KUKA KRL program: MyProgram_202().src

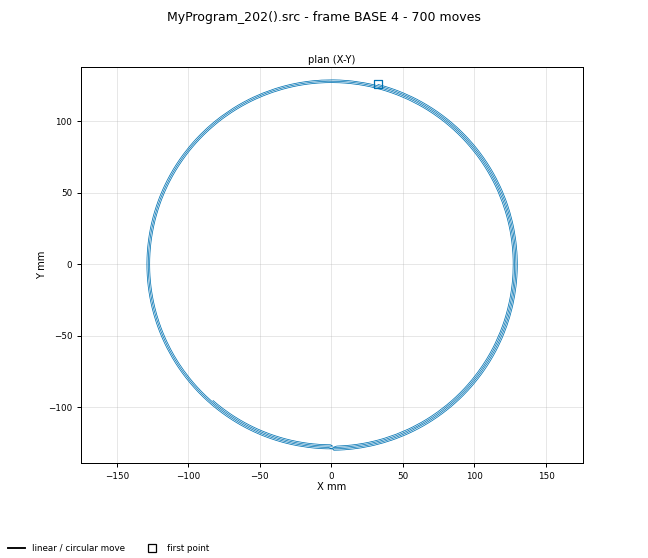
[picture p0: tool path of MyProgram_202().src in frame BASE 4, 700 of 700 moves have a stored position in this frame; points joined in program order, loops and branches not executed]
&ACCESS RVP
&REL 1
&PARAM TEMPLATE = C:\KRC\Roboter\Template\vorgabe
&PARAM EDITMASK = *
DEF MyProgram_202()
; ---- Setting reference (Base) ----
$BASE = BASE_DATA[4]

; --------------------------
; ---- Setting tool (TCP) ----
$TOOL = TOOL_DATA[3]
; --------------------------

$VEL.CP = VEL_APROX_PRINT
Startdeposition()
$VEL.CP = VEL_PRINT
LIN {X 32.4912,Y 125.808,Z 145,A 71.2576,B 24.9481,C -1.6638,E1 25.0411,E2 735.1147} C_DIS
LIN {X 35.4969,Y 124.993,Z 145,A 69.8884,B 24.9481,C -1.663,E1 25.0447,E2 736.4834} C_DIS
LIN {X 38.2252,Y 124.1849,Z 145,A 68.5665,B 24.9484,C -1.6587,E1 25.0483,E2 737.8133} C_DIS
LIN {X 41.3157,Y 123.1913,Z 145,A 67.1752,B 24.9484,C -1.6595,E1 25.052,E2 739.1999} C_DIS
LIN {X 44.3236,Y 122.1413,Z 145,A 65.7721,B 24.9484,C -1.6583,E1 25.0557,E2 740.6031} C_DIS
LIN {X 47.3297,Y 121.0081,Z 145,A 64.3243,B 24.9487,C -1.6553,E1 25.0595,E2 742.0548} C_DIS
LIN {X 50.4558,Y 119.7388,Z 145,A 62.8585,B 24.9487,C -1.6548,E1 25.0632,E2 743.5183} C_DIS
LIN {X 53.4411,Y 118.4365,Z 145,A 61.4515,B 24.9487,C -1.6547,E1 25.0668,E2 744.9223} C_DIS
LIN {X 56.2396,Y 117.133,Z 145,A 60.0583,B 24.9489,C -1.6514,E1 25.0703,E2 746.3197} C_DIS
LIN {X 59.4678,Y 115.5287,Z 145,A 58.4153,B 24.9492,C -1.6465,E1 25.0745,E2 747.9697} C_DIS
LIN {X 63.2279,Y 113.5157,Z 145,A 56.501,B 24.9495,C -1.6421,E1 25.0792,E2 749.8887} C_DIS
LIN {X 66.9845,Y 111.3401,Z 145,A 54.5775,B 24.9497,C -1.6388,E1 25.0838,E2 751.8143} C_DIS
LIN {X 70.8468,Y 108.923,Z 145,A 52.626,B 24.9497,C -1.6385,E1 25.0884,E2 753.76} C_DIS
LIN {X 74.4541,Y 106.4901,Z 145,A 50.7053,B 24.9499,C -1.6352,E1 25.0928,E2 755.6822} C_DIS
LIN {X 77.9363,Y 103.9691,Z 145,A 48.7841,B 24.9502,C -1.6304,E1 25.0971,E2 757.6077} C_DIS
LIN {X 81.3309,Y 101.3353,Z 145,A 46.8925,B 24.9504,C -1.627,E1 25.1013,E2 759.5003} C_DIS
LIN {X 84.4776,Y 98.7278,Z 145,A 45.1201,B 24.9505,C -1.625,E1 25.1051,E2 761.2706} C_DIS
LIN {X 87.6247,Y 95.9456,Z 145,A 43.3009,B 24.9506,C -1.6229,E1 25.1088,E2 763.0875} C_DIS
LIN {X 90.595,Y 93.1456,Z 145,A 41.5081,B 24.9509,C -1.6195,E1 25.1124,E2 764.881} C_DIS
LIN {X 93.6458,Y 90.0783,Z 145,A 39.6489,B 24.9509,C -1.6178,E1 25.1161,E2 766.7363} C_DIS
LIN {X 96.4286,Y 87.0923,Z 145,A 37.8481,B 24.9512,C -1.6136,E1 25.1195,E2 768.539} C_DIS
LIN {X 99.1768,Y 83.9494,Z 145,A 36.042,B 24.9514,C -1.6111,E1 25.1228,E2 770.3429} C_DIS
LIN {X 101.4035,Y 81.2464,Z 145,A 34.4908,B 24.9516,C -1.607,E1 25.1255,E2 771.8966} C_DIS
LIN {X 103.8668,Y 78.0719,Z 145,A 32.6881,B 24.952,C -1.6009,E1 25.1286,E2 773.705} C_DIS
LIN {X 106.4211,Y 74.5532,Z 145,A 30.7475,B 24.9523,C -1.5948,E1 25.1317,E2 775.6507} C_DIS
LIN {X 108.7748,Y 71.075,Z 145,A 28.8761,B 24.9527,C -1.5889,E1 25.1346,E2 777.5267} C_DIS
LIN {X 111.0977,Y 67.3855,Z 145,A 27.0107,B 24.9528,C -1.5867,E1 25.1374,E2 779.3877} C_DIS
LIN {X 113.2935,Y 63.6243,Z 145,A 25.1416,B 24.953,C -1.5841,E1 25.14,E2 781.2532} C_DIS
LIN {X 115.2071,Y 60.0868,Z 145,A 23.4203,B 24.9531,C -1.5819,E1 25.1422,E2 782.9706} C_DIS
LIN {X 116.7275,Y 57.0777,Z 145,A 21.9744,B 24.9532,C -1.5798,E1 25.144,E2 784.4138} C_DIS
LIN {X 118.0523,Y 54.2836,Z 145,A 20.5723,B 24.9536,C -1.5738,E1 25.1457,E2 785.8224} C_DIS
LIN {X 119.393,Y 51.2678,Z 145,A 19.1594,B 24.9537,C -1.5718,E1 25.1472,E2 787.2323} C_DIS
LIN {X 120.7266,Y 48.0458,Z 145,A 17.6476,B 24.9539,C -1.5686,E1 25.1488,E2 788.7434} C_DIS
LIN {X 121.789,Y 45.2829,Z 145,A 16.3455,B 24.9541,C -1.5649,E1 25.1501,E2 790.0471} C_DIS
LIN {X 122.9304,Y 42.0878,Z 145,A 14.8729,B 24.9543,C -1.5615,E1 25.1515,E2 791.5193} C_DIS
LIN {X 124.0143,Y 38.7826,Z 145,A 13.332,B 24.9546,C -1.5564,E1 25.1528,E2 793.0634} C_DIS
LIN {X 124.7733,Y 36.2591,Z 145,A 12.1683,B 24.9548,C -1.5528,E1 25.1537,E2 794.2291} C_DIS
LIN {X 125.6228,Y 33.1968,Z 145,A 10.7859,B 24.955,C -1.5494,E1 25.1547,E2 795.6116} C_DIS
LIN {X 126.3733,Y 30.2137,Z 145,A 9.4857,B 24.955,C -1.5481,E1 25.1556,E2 796.9072} C_DIS
LIN {X 127.0123,Y 27.403,Z 145,A 8.1592,B 24.9555,C -1.5411,E1 25.1564,E2 798.2425} C_DIS
LIN {X 127.6864,Y 24.0695,Z 145,A 6.6754,B 24.9557,C -1.5372,E1 25.1572,E2 799.727} C_DIS
LIN {X 128.2522,Y 20.8498,Z 145,A 5.2557,B 24.9559,C -1.5337,E1 25.1579,E2 801.1466} C_DIS
LIN {X 128.7042,Y 17.8487,Z 145,A 3.9702,B 24.956,C -1.5322,E1 25.1584,E2 802.428} C_DIS
LIN {X 129.0189,Y 15.4011,Z 145,A 2.831,B 24.9564,C -1.5259,E1 25.1588,E2 803.5752} C_DIS
LIN {X 129.3909,Y 11.89,Z 145,A 1.3171,B 24.9565,C -1.5231,E1 25.1592,E2 805.0868} C_DIS
LIN {X 129.6283,Y 8.9369,Z 145,A 0.0617,B 24.9566,C -1.5216,E1 25.1595,E2 806.3383} C_DIS
LIN {X 129.7846,Y 6.2559,Z 145,A -1.1949,B 24.9571,C -1.5138,E1 25.1596,E2 807.6058} C_DIS
LIN {X 129.9157,Y 2.2459,Z 145,A -2.9323,B 24.9573,C -1.5097,E1 25.1598,E2 809.3425} C_DIS
LIN {X 129.9256,Y -1.648,Z 145,A -4.7087,B 24.9578,C -1.5008,E1 25.1598,E2 811.1293} C_DIS
LIN {X 129.8316,Y -5.1857,Z 145,A -6.2154,B 24.9579,C -1.4986,E1 25.1596,E2 812.6323} C_DIS
LIN {X 129.6439,Y -8.7237,Z 145,A -7.7185,B 24.958,C -1.4966,E1 25.1594,E2 814.1312} C_DIS
LIN {X 129.3753,Y -12.0517,Z 145,A -9.2549,B 24.9585,C -1.4883,E1 25.159,E2 815.678} C_DIS
LIN {X 129.012,Y -15.4589,Z 145,A -10.7277,B 24.9587,C -1.4853,E1 25.1585,E2 817.1491} C_DIS
LIN {X 128.5211,Y -19.1304,Z 145,A -12.3114,B 24.9588,C -1.4826,E1 25.1579,E2 818.73} C_DIS
LIN {X 128.0736,Y -21.9207,Z 145,A -13.5064,B 24.9588,C -1.4813,E1 25.1574,E2 819.9211} C_DIS
LIN {X 127.6134,Y -24.4517,Z 145,A -14.6895,B 24.9592,C -1.4749,E1 25.1568,E2 821.1122} C_DIS
LIN {X 126.9339,Y -27.7659,Z 145,A -16.1647,B 24.9595,C -1.4709,E1 25.1559,E2 822.5881} C_DIS
LIN {X 126.2492,Y -30.7286,Z 145,A -17.4909,B 24.9597,C -1.4673,E1 25.1551,E2 823.9151} C_DIS
LIN {X 125.4352,Y -33.9003,Z 145,A -18.9313,B 24.9599,C -1.4628,E1 25.154,E2 825.3578} C_DIS
LIN {X 124.6228,Y -36.7728,Z 145,A -20.2611,B 24.9602,C -1.4579,E1 25.153,E2 826.6918} C_DIS
LIN {X 123.6135,Y -40.0371,Z 145,A -21.7437,B 24.9604,C -1.4543,E1 25.1518,E2 828.1744} C_DIS
LIN {X 122.6529,Y -42.888,Z 145,A -23.0454,B 24.9605,C -1.4514,E1 25.1506,E2 829.4756} C_DIS
LIN {X 121.5617,Y -45.8895,Z 145,A -24.4397,B 24.9607,C -1.4477,E1 25.1492,E2 830.8707} C_DIS
LIN {X 120.4111,Y -48.8285,Z 145,A -25.8611,B 24.9611,C -1.4417,E1 25.1478,E2 832.2984} C_DIS
LIN {X 119.0356,Y -52.0946,Z 145,A -27.3824,B 24.9612,C -1.439,E1 25.1461,E2 833.8176} C_DIS
LIN {X 117.594,Y -55.2747,Z 145,A -28.9303,B 24.9615,C -1.4338,E1 25.1443,E2 835.3695} C_DIS
LIN {X 116.4176,Y -57.7059,Z 145,A -30.1387,B 24.9617,C -1.4293,E1 25.1428,E2 836.5822} C_DIS
LIN {X 115.017,Y -60.4488,Z 145,A -31.4457,B 24.9618,C -1.4279,E1 25.1411,E2 837.8855} C_DIS
LIN {X 113.0688,Y -64.0241,Z 145,A -33.3523,B 24.9624,C -1.4165,E1 25.1385,E2 839.809} C_DIS
LIN {X 110.9386,Y -67.6478,Z 145,A -35.2233,B 24.9628,C -1.4101,E1 25.1358,E2 841.6854} C_DIS
LIN {X 108.7567,Y -71.1028,Z 145,A -36.8864,B 24.9626,C -1.4123,E1 25.1333,E2 843.3351} C_DIS
LIN {X 106.8976,Y -73.8683,Z 145,A -38.3473,B 24.9628,C -1.4086,E1 25.131,E2 844.7976} C_DIS
LIN {X 104.8526,Y -76.7427,Z 145,A -39.995,B 24.9633,C -1.3993,E1 25.1283,E2 846.4591} C_DIS
LIN {X 102.2417,Y -80.1879,Z 145,A -41.8596,B 24.9635,C -1.3962,E1 25.1251,E2 848.3222} C_DIS
LIN {X 99.8885,Y -83.1014,Z 145,A -43.4331,B 24.9635,C -1.3959,E1 25.1224,E2 849.889} C_DIS
LIN {X 97.7073,Y -85.6553,Z 145,A -44.9059,B 24.9637,C -1.3925,E1 25.1197,E2 851.3634} C_DIS
LIN {X 95.2327,Y -88.3982,Z 145,A -46.6386,B 24.9642,C -1.3827,E1 25.1164,E2 853.1114} C_DIS
LIN {X 92.0534,Y -91.7042,Z 145,A -48.5566,B 24.9642,C -1.3832,E1 25.1126,E2 855.0202} C_DIS
LIN {X 89.4704,Y -94.2268,Z 145,A -50.1556,B 24.9644,C -1.3789,E1 25.1094,E2 856.6226} C_DIS
LIN {X 86.4321,Y -97.021,Z 145,A -52.0108,B 24.9647,C -1.3727,E1 25.1056,E2 858.485} C_DIS
LIN {X 83.2465,Y -99.7678,Z 145,A -53.7858,B 24.9647,C -1.3727,E1 25.1018,E2 860.2532} C_DIS
LIN {X 80.5905,Y -101.9255,Z 145,A -55.2797,B 24.9648,C -1.37,E1 25.0986,E2 861.7477} C_DIS
LIN {X 77.5468,Y -104.2591,Z 145,A -57.0149,B 24.9651,C -1.364,E1 25.0947,E2 863.4907} C_DIS
LIN {X 74.0334,Y -106.7828,Z 145,A -58.9095,B 24.9653,C -1.3607,E1 25.0903,E2 865.3865} C_DIS
LIN {X 70.5061,Y -109.1441,Z 145,A -60.7379,B 24.9653,C -1.3592,E1 25.0861,E2 867.2124} C_DIS
LIN {X 67.5911,Y -110.9734,Z 145,A -62.3516,B 24.9658,C -1.3512,E1 25.0822,E2 868.8399} C_DIS
LIN {X 63.857,Y -113.1627,Z 145,A -64.2476,B 24.9659,C -1.3484,E1 25.0776,E2 870.7369} C_DIS
LIN {X 59.89,Y -115.3104,Z 145,A -66.1258,B 24.9659,C -1.3507,E1 25.073,E2 872.6042} C_DIS
LIN {X 57.2655,Y -116.6348,Z 145,A -67.4291,B 24.9659,C -1.3482,E1 25.0698,E2 873.91} C_DIS
LIN {X 54.009,Y -118.1792,Z 145,A -68.987,B 24.966,C -1.3473,E1 25.0658,E2 875.4662} C_DIS
LIN {X 51.1346,Y -119.4506,Z 145,A -70.3453,B 24.966,C -1.3466,E1 25.0624,E2 876.8227} C_DIS
LIN {X 48.119,Y -120.6971,Z 145,A -71.7959,B 24.9662,C -1.3439,E1 25.0586,E2 878.2764} C_DIS
LIN {X 45.203,Y -121.8189,Z 145,A -73.1449,B 24.9662,C -1.3435,E1 25.0551,E2 879.6235} C_DIS
LIN {X 42.4199,Y -122.8152,Z 145,A -74.4837,B 24.9664,C -1.3399,E1 25.0515,E2 880.968} C_DIS
LIN {X 39.0302,Y -123.9352,Z 145,A -76.0399,B 24.9664,C -1.3389,E1 25.0474,E2 882.5237} C_DIS
LIN {X 36.2163,Y -124.7858,Z 145,A -77.3172,B 24.9664,C -1.3384,E1 25.044,E2 883.8} C_DIS
LIN {X 33.1812,Y -125.6269,Z 145,A -78.7387,B 24.9666,C -1.3352,E1 25.0401,E2 885.2268} C_DIS
LIN {X 30.2349,Y -126.3682,Z 145,A -80.0521,B 24.9666,C -1.3352,E1 25.0366,E2 886.5383} C_DIS
LIN {X 27.2585,Y -127.0435,Z 145,A -81.4363,B 24.9668,C -1.3319,E1 25.0328,E2 887.9283} C_DIS
LIN {X 23.6437,Y -127.7678,Z 145,A -83.0096,B 24.9668,C -1.3332,E1 25.0285,E2 889.4968} C_DIS
LIN {X 20.8498,Y -128.2522,Z 145,A -84.2663,B 24.9668,C -1.3319,E1 25.025,E2 890.7552} C_DIS
LIN {X 17.8487,Y -128.7042,Z 145,A -85.6004,B 24.9668,C -1.3312,E1 25.0213,E2 892.0898} C_DIS
LIN {X 14.8613,Y -129.0833,Z 145,A -86.924,B 24.9668,C -1.3306,E1 25.0177,E2 893.4139} C_DIS
LIN {X 11.89,Y -129.3909,Z 145,A -88.192,B 24.9668,C -1.3324,E1 25.0142,E2 894.6769} C_DIS
LIN {X 9.2153,Y -129.608,Z 145,A -89.4167,B 24.9668,C -1.3297,E1 25.0107,E2 895.9073} C_DIS
LIN {X 5.3463,Y -129.8253,Z 145,A -91.179,B 24.9671,C -1.3263,E1 25.0058,E2 897.6771} C_DIS
LIN {X 1.648,Y -129.9256,Z 145,A -92.7481,B 24.9669,C -1.3289,E1 25.0014,E2 899.2396} C_DIS
LIN {X 1.648,Y -129.9256,Z 145,A -92.7481,B 24.9669,C -1.3289,E1 25.0014,E2 899.2396} C_DIS
Enddeposition()
LIN {X 0.9172,Y -128.9653,Z 145,A -92.8374,B 24.5098,C -1.2621,E1 24.5412,E2 899.4275} C_DIS
Startdeposition()
$VEL.CP = VEL_PRINT
LIN {X 5.042,Y -128.8762,Z 145,A -90.5283,B 24.5086,C -1.2863,E1 24.5478,E2 897.0606} C_DIS
LIN {X 8.2974,Y -128.7081,Z 145,A -88.9865,B 24.5084,C -1.2916,E1 24.5521,E2 895.5066} C_DIS
LIN {X 12.5181,Y -128.3659,Z 145,A -87.1558,B 24.5084,C -1.29,E1 24.5572,E2 893.6807} C_DIS
LIN {X 18.1324,Y -127.6937,Z 145,A -84.5266,B 24.5081,C -1.2976,E1 24.5645,E2 891.0355} C_DIS
LIN {X 22.5529,Y -126.9876,Z 145,A -82.639,B 24.5083,C -1.294,E1 24.5697,E2 889.1586} C_DIS
LIN {X 26.1324,Y -126.3001,Z 145,A -80.9242,B 24.5079,C -1.3002,E1 24.5744,E2 887.4308} C_DIS
LIN {X 30.1447,Y -125.4023,Z 145,A -79.2248,B 24.5082,C -1.2955,E1 24.579,E2 885.7451} C_DIS
LIN {X 33.3745,Y -124.5816,Z 145,A -77.7418,B 24.5081,C -1.2972,E1 24.583,E2 884.2605} C_DIS
LIN {X 37.1134,Y -123.521,Z 145,A -75.7574,B 24.5073,C -1.3124,E1 24.5884,E2 882.2431} C_DIS
LIN {X 42.3908,Y -121.809,Z 145,A -73.5836,B 24.5079,C -1.3006,E1 24.5941,E2 880.1019} C_DIS
LIN {X 45.7996,Y -120.5701,Z 145,A -71.8309,B 24.5075,C -1.31,E1 24.5987,E2 878.3304} C_DIS
LIN {X 49.5713,Y -119.0676,Z 145,A -69.8378,B 24.5068,C -1.3224,E1 24.6039,E2 876.3122} C_DIS
LIN {X 52.6398,Y -117.743,Z 145,A -68.6461,B 24.5075,C -1.3096,E1 24.6069,E2 875.1542} C_DIS
LIN {X 56.4236,Y -115.9795,Z 145,A -66.7297,B 24.5072,C -1.3157,E1 24.6118,E2 873.2281} C_DIS
LIN {X 65.6898,Y -110.9946,Z 145,A -62.1749,B 24.5071,C -1.3177,E1 24.6229,E2 868.6821} C_DIS
LIN {X 69.8564,Y -108.4208,Z 145,A -60.0132,B 24.5069,C -1.3212,E1 24.628,E2 866.5192} C_DIS
LIN {X 72.8158,Y -106.4554,Z 145,A -58.3755,B 24.5066,C -1.3275,E1 24.6318,E2 864.8719} C_DIS
LIN {X 76.1855,Y -104.0705,Z 145,A -56.501,B 24.5063,C -1.3334,E1 24.6361,E2 862.9898} C_DIS
LIN {X 79.4416,Y -101.6069,Z 145,A -54.6674,B 24.506,C -1.3384,E1 24.6401,E2 861.1511} C_DIS
LIN {X 82.3725,Y -99.2453,Z 145,A -53.098,B 24.506,C -1.3368,E1 24.6435,E2 859.5916} C_DIS
LIN {X 85.2992,Y -96.7416,Z 145,A -51.4153,B 24.506,C -1.3393,E1 24.647,E2 857.9097} C_DIS
LIN {X 88.2732,Y -94.0361,Z 145,A -49.5828,B 24.5056,C -1.3461,E1 24.6508,E2 856.0687} C_DIS
LIN {X 91.1569,Y -91.2436,Z 145,A -47.9186,B 24.5057,C -1.3442,E1 24.6541,E2 854.416} C_DIS
LIN {X 93.7338,Y -88.5936,Z 145,A -46.1682,B 24.5052,C -1.354,E1 24.6575,E2 852.6497} C_DIS
LIN {X 96.647,Y -85.4061,Z 145,A -44.3102,B 24.5052,C -1.3558,E1 24.661,E2 850.7959} C_DIS
LIN {X 99.348,Y -82.2485,Z 145,A -42.3389,B 24.5045,C -1.3674,E1 24.6646,E2 848.8061} C_DIS
LIN {X 102.2616,Y -78.5971,Z 145,A -40.3258,B 24.5044,C -1.3697,E1 24.668,E2 846.7971} C_DIS
LIN {X 104.9015,Y -75.0369,Z 145,A -38.2409,B 24.5038,C -1.3814,E1 24.6715,E2 844.6946} C_DIS
LIN {X 109.1864,Y -68.6522,Z 145,A -34.9427,B 24.5036,C -1.3849,E1 24.6765,E2 841.4047} C_DIS
LIN {X 111.0541,Y -65.5892,Z 145,A -33.3576,B 24.5034,C -1.3891,E1 24.6788,E2 839.8179} C_DIS
LIN {X 113.3781,Y -61.4847,Z 145,A -31.3272,B 24.5032,C -1.3919,E1 24.6815,E2 837.7915} C_DIS
LIN {X 115.0369,Y -58.3174,Z 145,A -29.8444,B 24.5032,C -1.3911,E1 24.6834,E2 836.3185} C_DIS
LIN {X 116.7701,Y -54.7687,Z 145,A -27.7093,B 24.5019,C -1.4167,E1 24.686,E2 834.1339} C_DIS
LIN {X 118.2649,Y -51.4575,Z 145,A -26.7258,B 24.5034,C -1.3883,E1 24.687,E2 833.2241} C_DIS
LIN {X 119.0606,Y -49.588,Z 145,A -25.6136,B 24.5027,C -1.4022,E1 24.6883,E2 832.0848} C_DIS
LIN {X 120.3938,Y -46.2598,Z 145,A -23.9046,B 24.5021,C -1.4133,E1 24.69,E2 830.3587} C_DIS
LIN {X 122.2439,Y -41.1214,Z 145,A -21.7994,B 24.5026,C -1.404,E1 24.6919,E2 828.2879} C_DIS
LIN {X 123.0704,Y -38.5821,Z 145,A -20.2512,B 24.5013,C -1.4269,E1 24.6933,E2 826.6937} C_DIS
LIN {X 124.2424,Y -34.6157,Z 145,A -18.6205,B 24.5016,C -1.4219,E1 24.6945,E2 825.0846} C_DIS
LIN {X 125.2378,Y -30.8269,Z 145,A -16.794,B 24.501,C -1.4321,E1 24.6958,E2 823.2445} C_DIS
LIN {X 126.0851,Y -27.1474,Z 145,A -15.2551,B 24.5011,C -1.4302,E1 24.6967,E2 821.7191} C_DIS
LIN {X 126.7255,Y -23.982,Z 145,A -13.7893,B 24.5008,C -1.4366,E1 24.6975,E2 820.2469} C_DIS
LIN {X 127.4291,Y -19.9072,Z 145,A -10.7727,B 24.4969,C -1.5058,E1 24.6989,E2 817.0823} C_DIS
LIN {X 128.4003,Y -12.1599,Z 145,A -8.7524,B 24.5006,C -1.4396,E1 24.6994,E2 815.233} C_DIS
LIN {X 128.6857,Y -8.6592,Z 145,A -6.7679,B 24.4991,C -1.4672,E1 24.6998,E2 813.1944} C_DIS
LIN {X 128.9118,Y -4.058,Z 145,A -4.8212,B 24.4991,C -1.4686,E1 24.7,E2 811.2561} C_DIS
LIN {X 128.9762,Y 0.3437,Z 145,A -2.8995,B 24.4988,C -1.4732,E1 24.7,E2 809.3351} C_DIS
LIN {X 128.758,Y 7.4881,Z 145,A 0.0508,B 24.4988,C -1.4717,E1 24.6998,E2 806.4064} C_DIS
LIN {X 128.2242,Y 13.8938,Z 145,A 3.0101,B 24.498,C -1.4864,E1 24.699,E2 803.4297} C_DIS
LIN {X 127.7263,Y 17.9044,Z 145,A 4.5867,B 24.4983,C -1.4806,E1 24.6985,E2 801.8765} C_DIS
LIN {X 127.3111,Y 20.6556,Z 145,A 6.0944,B 24.4973,C -1.4989,E1 24.6978,E2 800.3339} C_DIS
LIN {X 126.6844,Y 24.1973,Z 145,A 7.5774,B 24.4973,C -1.498,E1 24.697,E2 798.862} C_DIS
LIN {X 125.9668,Y 27.6953,Z 145,A 9.2816,B 24.4967,C -1.5092,E1 24.696,E2 797.141} C_DIS
LIN {X 125.0296,Y 31.6546,Z 145,A 10.9355,B 24.4968,C -1.5068,E1 24.6949,E2 795.5027} C_DIS
LIN {X 124.1886,Y 34.8083,Z 145,A 12.3832,B 24.4966,C -1.5112,E1 24.6939,E2 794.0529} C_DIS
LIN {X 123.1959,Y 38.1755,Z 145,A 14.0747,B 24.4959,C -1.523,E1 24.6925,E2 792.3431} C_DIS
LIN {X 121.8051,Y 42.402,Z 145,A 15.9011,B 24.496,C -1.5211,E1 24.6909,E2 790.5318} C_DIS
LIN {X 120.7475,Y 45.3258,Z 145,A 17.277,B 24.4958,C -1.5249,E1 24.6895,E2 789.1544} C_DIS
LIN {X 119.3674,Y 48.8493,Z 145,A 19.2308,B 24.4946,C -1.5443,E1 24.6875,E2 787.1653} C_DIS
LIN {X 117.5648,Y 53.0382,Z 145,A 20.9232,B 24.4953,C -1.5327,E1 24.6856,E2 785.5102} C_DIS
LIN {X 116.3389,Y 55.6743,Z 145,A 22.2306,B 24.4951,C -1.5372,E1 24.684,E2 784.199} C_DIS
LIN {X 114.7641,Y 58.8533,Z 145,A 23.8574,B 24.4946,C -1.5443,E1 24.682,E2 782.564} C_DIS
LIN {X 112.6959,Y 62.7261,Z 145,A 25.9472,B 24.4939,C -1.557,E1 24.6791,E2 780.4549} C_DIS
LIN {X 110.1549,Y 67.0888,Z 145,A 28.1143,B 24.4938,C -1.5592,E1 24.6761,E2 778.294} C_DIS
LIN {X 108.2811,Y 70.072,Z 145,A 29.6406,B 24.4936,C -1.5613,E1 24.6738,E2 776.7705} C_DIS
LIN {X 105.8567,Y 73.6831,Z 145,A 31.5435,B 24.4934,C -1.5648,E1 24.6708,E2 774.8688} C_DIS
LIN {X 103.2464,Y 77.2991,Z 145,A 33.4979,B 24.4932,C -1.5684,E1 24.6675,E2 772.9154} C_DIS
LIN {X 100.8045,Y 80.4571,Z 145,A 35.2068,B 24.4932,C -1.5694,E1 24.6646,E2 771.2121} C_DIS
LIN {X 98.543,Y 83.2124,Z 145,A 36.8806,B 24.4926,C -1.5779,E1 24.6616,E2 769.5259} C_DIS
LIN {X 95.7514,Y 86.4097,Z 145,A 39.3329,B 24.4906,C -1.6117,E1 24.6569,E2 767.0034} C_DIS
LIN {X 92.2184,Y 90.1699,Z 145,A 40.9534,B 24.4924,C -1.5819,E1 24.6539,E2 765.4616} C_DIS
LIN {X 89.338,Y 93.0251,Z 145,A 42.8345,B 24.4919,C -1.5899,E1 24.6501,E2 763.5695} C_DIS
LIN {X 86.0756,Y 96.0512,Z 145,A 44.7867,B 24.4917,C -1.5927,E1 24.6461,E2 761.6186} C_DIS
LIN {X 82.823,Y 98.8697,Z 145,A 46.6014,B 24.4918,C -1.5915,E1 24.6422,E2 759.814} C_DIS
LIN {X 79.9093,Y 101.2395,Z 145,A 48.3383,B 24.4914,C -1.5981,E1 24.6384,E2 758.0677} C_DIS
LIN {X 76.5354,Y 103.8134,Z 145,A 50.2418,B 24.4911,C -1.6025,E1 24.6342,E2 756.1607} C_DIS
LIN {X 73.1048,Y 106.257,Z 145,A 52.1163,B 24.4909,C -1.6059,E1 24.6299,E2 754.2848} C_DIS
LIN {X 69.2727,Y 108.7945,Z 145,A 54.192,B 24.4906,C -1.6109,E1 24.625,E2 752.2039} C_DIS
LIN {X 65.331,Y 111.2057,Z 145,A 56.2125,B 24.4906,C -1.6124,E1 24.6202,E2 750.1862} C_DIS
LIN {X 61.4184,Y 113.4143,Z 145,A 58.1643,B 24.4905,C -1.613,E1 24.6154,E2 748.2388} C_DIS
LIN {X 58.3822,Y 115.0039,Z 145,A 59.5685,B 24.4907,C -1.609,E1 24.6119,E2 746.8481} C_DIS
LIN {X 55.3148,Y 116.5107,Z 145,A 61.0639,B 24.4907,C -1.6098,E1 24.6082,E2 745.3548} C_DIS
LIN {X 52.5043,Y 117.8036,Z 145,A 62.4741,B 24.4905,C -1.6132,E1 24.6046,E2 743.94} C_DIS
LIN {X 48.9828,Y 119.3133,Z 145,A 64.142,B 24.4905,C -1.6133,E1 24.6003,E2 742.2758} C_DIS
LIN {X 45.0791,Y 120.8399,Z 145,A 66.0297,B 24.4903,C -1.6165,E1 24.5954,E2 740.3847} C_DIS
LIN {X 41.5737,Y 122.0923,Z 145,A 67.8767,B 24.4896,C -1.6276,E1 24.5904,E2 738.5146} C_DIS
LIN {X 37.3576,Y 123.4462,Z 145,A 69.6419,B 24.4901,C -1.6191,E1 24.5858,E2 736.7733} C_DIS
LIN {X 33.4874,Y 124.5515,Z 145,A 71.4784,B 24.4899,C -1.6227,E1 24.5808,E2 734.9311} C_DIS
LIN {X 30.2084,Y 125.3869,Z 145,A 72.9173,B 24.49,C -1.6205,E1 24.577,E2 733.4998} C_DIS
LIN {X 26.7242,Y 126.1765,Z 145,A 74.6365,B 24.4896,C -1.6278,E1 24.5722,E2 731.7653} C_DIS
LIN {X 22.7495,Y 126.9524,Z 145,A 76.3137,B 24.4899,C -1.6225,E1 24.5677,E2 730.1026} C_DIS
LIN {X 14.6498,Y 128.1407,Z 145,A 79.8929,B 24.49,C -1.6205,E1 24.5578,E2 726.5314} C_DIS
LIN {X 11.5908,Y 128.4549,Z 145,A 82.1032,B 24.4874,C -1.6624,E1 24.5514,E2 724.2215} C_DIS
LIN {X 5.9542,Y 128.8383,Z 145,A 83.6204,B 24.4905,C -1.6134,E1 24.5475,E2 722.8229} C_DIS
LIN {X 1.2351,Y 128.97,Z 145,A 85.7882,B 24.4903,C -1.6166,E1 24.5414,E2 720.648} C_DIS
LIN {X -6.7547,Y 128.7981,Z 145,A 89.0228,B 24.4913,C -1.6003,E1 24.5325,E2 717.4524} C_DIS
LIN {X -12.9942,Y 128.3202,Z 145,A 92.2107,B 24.4901,C -1.6186,E1 24.5235,E2 714.2189} C_DIS
LIN {X -17.1637,Y 127.8282,Z 145,A 93.9613,B 24.4906,C -1.612,E1 24.5187,E2 712.483} C_DIS
LIN {X -21.508,Y 127.1689,Z 145,A 96.1698,B 24.4899,C -1.623,E1 24.5125,E2 710.2459} C_DIS
LIN {X -25.6277,Y 126.4028,Z 145,A 97.9479,B 24.4902,C -1.6174,E1 24.5076,E2 708.4792} C_DIS
LIN {X -29.0652,Y 125.6573,Z 145,A 99.4905,B 24.4904,C -1.6151,E1 24.5035,E2 706.9404} C_DIS
LIN {X -32.9269,Y 124.701,Z 145,A 101.3188,B 24.4903,C -1.6162,E1 24.4985,E2 705.1065} C_DIS
LIN {X -36.2257,Y 123.7825,Z 145,A 102.967,B 24.49,C -1.6206,E1 24.494,E2 703.4449} C_DIS
LIN {X -39.6757,Y 122.721,Z 145,A 104.4442,B 24.4905,C -1.6127,E1 24.4901,E2 701.9842} C_DIS
LIN {X -47.9038,Y 119.7486,Z 145,A 108.1068,B 24.4915,C -1.5969,E1 24.4807,E2 698.3522} C_DIS
LIN {X -51.8029,Y 118.1156,Z 145,A 110.1507,B 24.4912,C -1.602,E1 24.4753,E2 696.2913} C_DIS
LIN {X -54.2774,Y 116.9972,Z 145,A 111.415,B 24.4912,C -1.6029,E1 24.4721,E2 695.0215} C_DIS
LIN {X -57.4019,Y 115.4969,Z 145,A 113.0392,B 24.491,C -1.6044,E1 24.468,E2 693.3895} C_DIS
LIN {X -61.4187,Y 113.4141,Z 145,A 115.0716,B 24.4912,C -1.602,E1 24.463,E2 691.357} C_DIS
LIN {X -65.156,Y 111.3085,Z 145,A 116.9543,B 24.4914,C -1.5975,E1 24.4585,E2 689.4796} C_DIS
LIN {X -68.7299,Y 109.1379,Z 145,A 118.8477,B 24.4916,C -1.5956,E1 24.454,E2 687.5845} C_DIS
LIN {X -76.9525,Y 103.5045,Z 145,A 123.2535,B 24.4922,C -1.5855,E1 24.4439,E2 683.1879} C_DIS
LIN {X -81.2776,Y 100.1446,Z 145,A 125.5991,B 24.4927,C -1.5761,E1 24.4388,E2 680.8562} C_DIS
LIN {X -83.4318,Y 98.3565,Z 145,A 126.9796,B 24.4925,C -1.5797,E1 24.4358,E2 679.4616} C_DIS
LIN {X -86.7662,Y 95.428,Z 145,A 128.9604,B 24.4928,C -1.5755,E1 24.4317,E2 677.4829} C_DIS
LIN {X -91.3941,Y 91.0054,Z 145,A 132.3128,B 24.4918,C -1.5923,E1 24.4249,E2 674.0754} C_DIS
LIN {X -94.6097,Y 87.6582,Z 145,A 133.6661,B 24.4941,C -1.5541,E1 24.4225,E2 672.8085} C_DIS
LIN {X -96.6517,Y 85.4008,Z 145,A 135.2499,B 24.4936,C -1.5614,E1 24.4195,E2 671.2} C_DIS
LIN {X -98.9924,Y 82.6767,Z 145,A 136.9366,B 24.4936,C -1.5614,E1 24.4164,E2 669.5054} C_DIS
LIN {X -103.4941,Y 76.9665,Z 145,A 139.9807,B 24.4947,C -1.544,E1 24.4113,E2 666.4885} C_DIS
LIN {X -105.6767,Y 73.9419,Z 145,A 141.7976,B 24.4945,C -1.5468,E1 24.4083,E2 664.6559} C_DIS
LIN {X -108.1203,Y 70.3198,Z 145,A 143.7155,B 24.4949,C -1.5402,E1 24.4054,E2 662.7442} C_DIS
LIN {X -110.4795,Y 66.5521,Z 145,A 145.7124,B 24.4952,C -1.5355,E1 24.4024,E2 660.7482} C_DIS
LIN {X -112.7692,Y 62.5938,Z 145,A 147.7645,B 24.4955,C -1.5305,E1 24.3996,E2 658.6974} C_DIS
LIN {X -114.8249,Y 58.7338,Z 145,A 149.6194,B 24.496,C -1.5206,E1 24.3972,E2 656.8562} C_DIS
LIN {X -116.44,Y 55.4628,Z 145,A 151.3161,B 24.4961,C -1.5192,E1 24.3952,E2 655.1535} C_DIS
LIN {X -117.8553,Y 52.3889,Z 145,A 152.7931,B 24.4965,C -1.5134,E1 24.3935,E2 653.6824} C_DIS
LIN {X -119.6999,Y 48.0246,Z 145,A 154.894,B 24.4968,C -1.5067,E1 24.3912,E2 651.5859} C_DIS
LIN {X -121.1059,Y 44.3642,Z 145,A 157.1484,B 24.4958,C -1.5247,E1 24.389,E2 649.2746} C_DIS
LIN {X -122.4718,Y 40.4371,Z 145,A 158.4617,B 24.4976,C -1.4944,E1 24.3879,E2 648.0273} C_DIS
LIN {X -123.7381,Y 36.3773,Z 145,A 160.1205,B 24.4985,C -1.4778,E1 24.3866,E2 646.399} C_DIS
LIN {X -124.6361,Y 33.1702,Z 145,A 161.8995,B 24.498,C -1.4867,E1 24.3852,E2 644.5878} C_DIS
LIN {X -125.849,Y 28.2259,Z 145,A 164.0818,B 24.4986,C -1.4758,E1 24.3838,E2 642.419} C_DIS
LIN {X -126.6875,Y 24.181,Z 145,A 166.0186,B 24.4986,C -1.4744,E1 24.3827,E2 640.4737} C_DIS
LIN {X -127.3406,Y 20.4791,Z 145,A 167.83,B 24.4986,C -1.4754,E1 24.3819,E2 638.6489} C_DIS
LIN {X -127.9135,Y 16.5125,Z 145,A 169.5828,B 24.499,C -1.4684,E1 24.3812,E2 636.9025} C_DIS
LIN {X -128.3767,Y 12.4062,Z 145,A 171.3656,B 24.4995,C -1.4599,E1 24.3807,E2 635.1294} C_DIS
LIN {X -128.7128,Y 8.2205,Z 145,A 173.2601,B 24.4998,C -1.4551,E1 24.3803,E2 633.2349} C_DIS
LIN {X -128.8897,Y 4.695,Z 145,A 174.9223,B 24.4998,C -1.4543,E1 24.3801,E2 631.5645} C_DIS
LIN {X -128.9766,Y 0.2825,Z 145,A 176.9131,B 24.5001,C -1.4492,E1 24.3801,E2 629.5736} C_DIS
LIN {X -128.9204,Y -3.7497,Z 145,A 178.6262,B 24.5006,C -1.4398,E1 24.3801,E2 627.8728} C_DIS
LIN {X -128.7379,Y -7.8144,Z 145,A -179.5753,B 24.501,C -1.4335,E1 24.3804,E2 626.0786} C_DIS
LIN {X -128.4223,Y -11.9313,Z 145,A -177.6933,B 24.5012,C -1.4297,E1 24.3809,E2 624.1942} C_DIS
LIN {X -128.0289,Y -15.5936,Z 145,A -176.1049,B 24.5016,C -1.4222,E1 24.3814,E2 622.6142} C_DIS
LIN {X -127.4859,Y -19.5404,Z 145,A -174.2927,B 24.5018,C -1.4185,E1 24.3821,E2 620.8001} C_DIS
LIN {X -126.8813,Y -23.1464,Z 145,A -172.5607,B 24.5018,C -1.4183,E1 24.383,E2 619.0582} C_DIS
LIN {X -126.0555,Y -27.2846,Z 145,A -170.8127,B 24.5024,C -1.4065,E1 24.3839,E2 617.3281} C_DIS
LIN {X -125.3211,Y -30.4815,Z 145,A -169.3025,B 24.5025,C -1.4044,E1 24.3849,E2 615.8141} C_DIS
LIN {X -124.1921,Y -34.7956,Z 145,A -167.3606,B 24.503,C -1.3964,E1 24.3863,E2 613.8799} C_DIS
LIN {X -122.4511,Y -40.4994,Z 145,A -164.7381,B 24.5035,C -1.387,E1 24.3885,E2 611.2649} C_DIS
LIN {X -121.3106,Y -43.7965,Z 145,A -163.0579,B 24.5035,C -1.3884,E1 24.3901,E2 609.5717} C_DIS
LIN {X -120.1746,Y -46.8237,Z 145,A -161.6835,B 24.5038,C -1.3812,E1 24.3914,E2 608.2066} C_DIS
LIN {X -118.9574,Y -49.8349,Z 145,A -160.2401,B 24.504,C -1.377,E1 24.393,E2 606.7653} C_DIS
LIN {X -117.6397,Y -52.8709,Z 145,A -158.7658,B 24.5042,C -1.3729,E1 24.3946,E2 605.2927} C_DIS
LIN {X -116.242,Y -55.8771,Z 145,A -157.2893,B 24.5044,C -1.3688,E1 24.3964,E2 603.8178} C_DIS
LIN {X -114.8322,Y -58.7195,Z 145,A -155.8311,B 24.5045,C -1.3671,E1 24.3982,E2 602.3558} C_DIS
LIN {X -112.5761,Y -62.9398,Z 145,A -153.7483,B 24.5049,C -1.3592,E1 24.401,E2 600.281} C_DIS
LIN {X -111.2843,Y -65.1973,Z 145,A -152.4391,B 24.5047,C -1.3632,E1 24.4029,E2 598.9551} C_DIS
LIN {X -108.8946,Y -69.1154,Z 145,A -150.3189,B 24.5048,C -1.3615,E1 24.406,E2 596.8279} C_DIS
LIN {X -106.8416,Y -72.2478,Z 145,A -148.7189,B 24.5052,C -1.3542,E1 24.4085,E2 595.2375} C_DIS
LIN {X -104.3479,Y -75.805,Z 145,A -146.7934,B 24.5055,C -1.3491,E1 24.4116,E2 593.3147} C_DIS
LIN {X -101.5028,Y -79.5741,Z 145,A -144.6753,B 24.5057,C -1.3449,E1 24.4152,E2 591.1965} C_DIS
LIN {X -98.7093,Y -83.0141,Z 145,A -142.6874,B 24.5059,C -1.3411,E1 24.4187,E2 589.2085} C_DIS
LIN {X -95.8541,Y -86.2957,Z 145,A -140.7723,B 24.5061,C -1.3358,E1 24.4223,E2 587.2973} C_DIS
LIN {X -92.9481,Y -89.4185,Z 145,A -138.8018,B 24.5061,C -1.3352,E1 24.4261,E2 585.3197} C_DIS
LIN {X -89.8477,Y -92.5326,Z 145,A -136.8699,B 24.5064,C -1.33,E1 24.4299,E2 583.3919} C_DIS
LIN {X -86.5091,Y -95.6612,Z 145,A -134.8513,B 24.5067,C -1.3252,E1 24.434,E2 581.3767} C_DIS
LIN {X -83.224,Y -98.5331,Z 145,A -132.8457,B 24.5067,C -1.3246,E1 24.4383,E2 579.3646} C_DIS
LIN {X -79.8125,Y -101.3156,Z 145,A -130.9168,B 24.507,C -1.3196,E1 24.4425,E2 577.4403} C_DIS
LIN {X -76.3135,Y -103.9765,Z 145,A -128.8863,B 24.507,C -1.3199,E1 24.4471,E2 575.4018} C_DIS
LIN {X -73.2788,Y -106.1376,Z 145,A -127.2716,B 24.5072,C -1.3151,E1 24.4507,E2 573.793} C_DIS
LIN {X -69.2228,Y -108.8265,Z 145,A -125.3771,B 24.508,C -1.2988,E1 24.4551,E2 571.9316} C_DIS
LIN {X -66.422,Y -110.5582,Z 145,A -123.8629,B 24.508,C -1.2991,E1 24.4587,E2 570.412} C_DIS
LIN {X -63.5278,Y -112.2462,Z 145,A -122.1638,B 24.5076,C -1.3071,E1 24.4629,E2 568.6884} C_DIS
LIN {X -59.9564,Y -114.191,Z 145,A -120.4393,B 24.5079,C -1.3007,E1 24.4671,E2 566.9744} C_DIS
LIN {X -56.8395,Y -115.7743,Z 145,A -118.9286,B 24.5081,C -1.2967,E1 24.4709,E2 565.4693} C_DIS
LIN {X -53.8342,Y -117.2022,Z 145,A -117.3629,B 24.508,C -1.2992,E1 24.4749,E2 563.8936} C_DIS
LIN {X -49.4988,Y -119.0978,Z 145,A -115.347,B 24.5083,C -1.2927,E1 24.48,E2 561.8885} C_DIS
LIN {X -46.4794,Y -120.3084,Z 145,A -113.8061,B 24.5082,C -1.296,E1 24.484,E2 560.3363} C_DIS
LIN {X -42.3093,Y -121.8373,Z 145,A -111.8642,B 24.5083,C -1.2927,E1 24.4891,E2 558.3984} C_DIS
LIN {X -38.9952,Y -122.9384,Z 145,A -110.2859,B 24.5083,C -1.2927,E1 24.4933,E2 556.817} C_DIS
LIN {X -34.6636,Y -124.229,Z 145,A -108.2985,B 24.5084,C -1.2904,E1 24.4987,E2 554.8321} C_DIS
LIN {X -31.195,Y -125.1463,Z 145,A -106.5988,B 24.5082,C -1.2946,E1 24.5033,E2 553.1197} C_DIS
LIN {X -27.3164,Y -126.0486,Z 145,A -104.9476,B 24.5086,C -1.2879,E1 24.5078,E2 551.4824} C_DIS
LIN {X -23.8675,Y -126.7474,Z 145,A -102.1881,B 24.5056,C -1.347,E1 24.5158,E2 548.5774} C_DIS
LIN {X -16.1862,Y -127.9563,Z 145,A -99.975,B 24.5087,C -1.284,E1 24.5215,E2 546.5144} C_DIS
LIN {X -11.7157,Y -128.4429,Z 145,A -98.0147,B 24.5088,C -1.2819,E1 24.5269,E2 544.5581} C_DIS
LIN {X -6.2687,Y -128.8225,Z 145,A -95.5794,B 24.5088,C -1.2825,E1 24.5337,E2 542.1207} C_DIS
LIN {X -2.9975,Y -128.9413,Z 145,A -93.9486,B 24.5084,C -1.2914,E1 24.5383,E2 540.468} C_DIS
LIN {X 0.9172,Y -128.9653,Z 145,A -92.8343,B 24.5099,C -1.2608,E1 24.5412,E2 539.4275} C_DIS
Enddeposition()
LIN {X 0.9172,Y -128.9653,Z 145,A -92.8343,B 24.5099,C -1.2608,E1 24.5412,E2 539.4275} C_DIS
Startdeposition()
$VEL.CP = VEL_PRINT
LIN {X -2.0484,Y -127.9982,Z 145,A -94.0159,B 23.6983,C -1.1212,E1 23.7202,E2 540.8446} C_DIS
LIN {X -7.2402,Y -127.8099,Z 145,A -96.3916,B 23.6983,C -1.1186,E1 23.7135,E2 543.2273} C_DIS
LIN {X -13.9475,Y -127.2526,Z 145,A -99.4935,B 23.6986,C -1.1146,E1 23.7049,E2 546.3408} C_DIS
LIN {X -19.4951,Y -126.5213,Z 145,A -102.1573,B 23.6989,C -1.1078,E1 23.6975,E2 549.0239} C_DIS
LIN {X -24.2237,Y -125.7017,Z 145,A -104.0784,B 23.6984,C -1.1191,E1 23.6923,E2 550.9189} C_DIS
LIN {X -28.2312,Y -124.8629,Z 145,A -105.907,B 23.6984,C -1.1201,E1 23.6873,E2 552.7473} C_DIS
LIN {X -31.3155,Y -124.125,Z 145,A -107.2784,B 23.6982,C -1.1231,E1 23.6836,E2 554.1132} C_DIS
LIN {X -34.4367,Y -123.2954,Z 145,A -108.7993,B 23.6983,C -1.1206,E1 23.6794,E2 555.6429} C_DIS
LIN {X -38.3026,Y -122.1516,Z 145,A -110.6838,B 23.6984,C -1.1182,E1 23.6744,E2 557.5368} C_DIS
LIN {X -41.5483,Y -121.0848,Z 145,A -112.4714,B 23.6989,C -1.1076,E1 23.6696,E2 559.3542} C_DIS
LIN {X -44.7803,Y -119.9265,Z 145,A -113.6535,B 23.6981,C -1.1253,E1 23.6666,E2 560.4949} C_DIS
LIN {X -48.3904,Y -118.5171,Z 145,A -115.7963,B 23.6988,C -1.1084,E1 23.6609,E2 562.685} C_DIS
LIN {X -51.7895,Y -117.0714,Z 145,A -117.0915,B 23.698,C -1.1265,E1 23.6577,E2 563.9382} C_DIS
LIN {X -55.0077,Y -115.5932,Z 145,A -118.6385,B 23.6979,C -1.1301,E1 23.6538,E2 565.4803} C_DIS
LIN {X -58.1624,Y -114.0383,Z 145,A -120.2045,B 23.6978,C -1.1325,E1 23.6499,E2 567.0448} C_DIS
LIN {X -61.211,Y -112.4336,Z 145,A -121.8386,B 23.6978,C -1.1303,E1 23.6458,E2 568.6892} C_DIS
LIN {X -65.1198,Y -110.2162,Z 145,A -123.9087,B 23.6978,C -1.1306,E1 23.6408,E2 570.7652} C_DIS
LIN {X -68.2388,Y -108.3123,Z 145,A -125.5664,B 23.6978,C -1.1321,E1 23.6369,E2 572.4246} C_DIS
LIN {X -72.1019,Y -105.7808,Z 145,A -127.4499,B 23.6973,C -1.1437,E1 23.6326,E2 574.2857} C_DIS
LIN {X -76.6326,Y -102.5455,Z 145,A -130.0733,B 23.6973,C -1.1421,E1 23.6266,E2 576.9229} C_DIS
LIN {X -80.0743,Y -99.8816,Z 145,A -132.1608,B 23.6975,C -1.1394,E1 23.622,E2 579.0253} C_DIS
LIN {X -83.8761,Y -96.711,Z 145,A -134.3166,B 23.6971,C -1.1464,E1 23.6174,E2 581.1726} C_DIS
LIN {X -87.239,Y -93.688,Z 145,A -136.3012,B 23.6969,C -1.1522,E1 23.6134,E2 583.151} C_DIS
LIN {X -90.4774,Y -90.5651,Z 145,A -138.3527,B 23.6968,C -1.1548,E1 23.6093,E2 585.2052} C_DIS
LIN {X -93.5052,Y -87.4352,Z 145,A -140.2886,B 23.6965,C -1.1597,E1 23.6055,E2 587.1377} C_DIS
LIN {X -96.3649,Y -84.2728,Z 145,A -142.1751,B 23.6963,C -1.165,E1 23.602,E2 589.0199} C_DIS
LIN {X -99.0241,Y -81.1315,Z 145,A -144.0327,B 23.6961,C -1.1687,E1 23.5987,E2 590.8775} C_DIS
LIN {X -103.3511,Y -75.5429,Z 145,A -147.2403,B 23.6958,C -1.1745,E1 23.5933,E2 594.0868} C_DIS
LIN {X -105.1928,Y -72.9561,Z 145,A -149.03,B 23.6964,C -1.162,E1 23.5904,E2 595.9171} C_DIS
LIN {X -107.3882,Y -69.684,Z 145,A -150.4428,B 23.6955,C -1.1819,E1 23.5883,E2 597.2876} C_DIS
LIN {X -109.7635,Y -65.8804,Z 145,A -152.4834,B 23.6953,C -1.1858,E1 23.5853,E2 599.3297} C_DIS
LIN {X -112.4641,Y -61.1547,Z 145,A -155.0381,B 23.6953,C -1.1873,E1 23.5818,E2 601.8949} C_DIS
LIN {X -114.6628,Y -56.9223,Z 145,A -156.9513,B 23.6945,C -1.2029,E1 23.5794,E2 603.7798} C_DIS
LIN {X -116.5177,Y -53.0267,Z 145,A -159.0652,B 23.6946,C -1.2004,E1 23.5769,E2 605.9121} C_DIS
LIN {X -118.0649,Y -49.4805,Z 145,A -160.6229,B 23.694,C -1.2131,E1 23.5752,E2 607.4473} C_DIS
LIN {X -119.2615,Y -46.5223,Z 145,A -162.144,B 23.694,C -1.2132,E1 23.5736,E2 608.9771} C_DIS
LIN {X -120.5243,Y -43.1462,Z 145,A -163.7477,B 23.6938,C -1.2184,E1 23.5721,E2 610.5773} C_DIS
LIN {X -122.3043,Y -37.8073,Z 145,A -166.4022,B 23.6937,C -1.2202,E1 23.5698,E2 613.2436} C_DIS
LIN {X -123.9189,Y -32.1276,Z 145,A -169.0312,B 23.6932,C -1.2289,E1 23.5679,E2 615.867} C_DIS
LIN {X -124.7955,Y -28.5261,Z 145,A -170.5508,B 23.6927,C -1.2401,E1 23.5669,E2 617.3679} C_DIS
LIN {X -125.4654,Y -25.4186,Z 145,A -172.0309,B 23.6926,C -1.2421,E1 23.566,E2 618.8524} C_DIS
LIN {X -126.2236,Y -21.3393,Z 145,A -173.9237,B 23.6924,C -1.2464,E1 23.5651,E2 620.7463} C_DIS
LIN {X -126.8149,Y -17.4946,Z 145,A -175.758,B 23.6924,C -1.2479,E1 23.5644,E2 622.5884} C_DIS
LIN {X -127.2805,Y -13.6884,Z 145,A -177.3828,B 23.6918,C -1.2574,E1 23.5639,E2 624.1998} C_DIS
LIN {X -127.6534,Y -9.6133,Z 145,A -179.24,B 23.6916,C -1.2622,E1 23.5634,E2 626.0569} C_DIS
LIN {X -127.8782,Y -5.9281,Z 145,A 179.0377,B 23.6915,C -1.2645,E1 23.5632,E2 627.7845} C_DIS
LIN {X -128,Y -1.9431,Z 145,A 177.2988,B 23.6911,C -1.2722,E1 23.5631,E2 629.515} C_DIS
LIN {X -127.9935,Y 2.3333,Z 145,A 175.3314,B 23.6909,C -1.2762,E1 23.5631,E2 631.4852} C_DIS
LIN {X -127.8563,Y 6.3629,Z 145,A 173.5714,B 23.6905,C -1.2839,E1 23.5633,E2 633.237} C_DIS
LIN {X -127.6121,Y 10.1608,Z 145,A 171.7666,B 23.6905,C -1.2851,E1 23.5637,E2 635.0504} C_DIS
LIN {X -127.2686,Y 13.799,Z 145,A 170.2036,B 23.69,C -1.2936,E1 23.5641,E2 636.6021} C_DIS
LIN {X -126.7636,Y 17.8534,Z 145,A 168.3818,B 23.6897,C -1.2998,E1 23.5648,E2 638.4199} C_DIS
LIN {X -126.2309,Y 21.2955,Z 145,A 166.7849,B 23.6895,C -1.3032,E1 23.5655,E2 640.0183} C_DIS
LIN {X -125.5028,Y 25.2347,Z 145,A 165.0261,B 23.6891,C -1.3104,E1 23.5664,E2 641.77} C_DIS
LIN {X -123.7195,Y 32.8809,Z 145,A 161.6628,B 23.6882,C -1.3281,E1 23.5686,E2 645.1098} C_DIS
LIN {X -121.8095,Y 39.3736,Z 145,A 158.4875,B 23.688,C -1.3314,E1 23.5711,E2 648.2965} C_DIS
LIN {X -120.8577,Y 42.2033,Z 145,A 157.016,B 23.6881,C -1.3297,E1 23.5724,E2 649.781} C_DIS
LIN {X -119.4576,Y 46.0179,Z 145,A 155.1925,B 23.6878,C -1.3352,E1 23.5742,E2 651.6019} C_DIS
LIN {X -117.0006,Y 51.948,Z 145,A 152.3498,B 23.6873,C -1.3453,E1 23.5773,E2 654.436} C_DIS
LIN {X -115.5818,Y 55.0315,Z 145,A 150.7756,B 23.6872,C -1.3475,E1 23.5792,E2 656.0137} C_DIS
LIN {X -114.0347,Y 58.1696,Z 145,A 149.2436,B 23.6868,C -1.3537,E1 23.5811,E2 657.539} C_DIS
LIN {X -112.6718,Y 60.7717,Z 145,A 147.6601,B 23.6873,C -1.3459,E1 23.5832,E2 659.1508} C_DIS
LIN {X -110.1296,Y 65.2662,Z 145,A 145.4516,B 23.6867,C -1.357,E1 23.5863,E2 661.3437} C_DIS
LIN {X -107.69,Y 69.2171,Z 145,A 143.3973,B 23.6863,C -1.364,E1 23.5893,E2 663.3916} C_DIS
LIN {X -105.3198,Y 72.7735,Z 145,A 141.4405,B 23.6861,C -1.3674,E1 23.5924,E2 665.3502} C_DIS
LIN {X -102.8207,Y 76.263,Z 145,A 139.5405,B 23.6858,C -1.3736,E1 23.5955,E2 667.2446} C_DIS
LIN {X -99.0854,Y 81.0566,Z 145,A 136.4882,B 23.6861,C -1.3665,E1 23.6009,E2 670.3299} C_DIS
LIN {X -96.6798,Y 83.9119,Z 145,A 135.2261,B 23.6849,C -1.3885,E1 23.6031,E2 671.5429} C_DIS
LIN {X -91.9262,Y 89.0935,Z 145,A 132.2466,B 23.6841,C -1.4037,E1 23.6087,E2 674.4984} C_DIS
LIN {X -87.7991,Y 93.1633,Z 145,A 129.5513,B 23.684,C -1.4054,E1 23.6141,E2 677.2013} C_DIS
LIN {X -82.9969,Y 97.4659,Z 145,A 126.0348,B 23.6852,C -1.3845,E1 23.6216,E2 680.7849} C_DIS
LIN {X -79.7625,Y 100.1301,Z 145,A 124.5832,B 23.6839,C -1.4071,E1 23.6246,E2 682.1858} C_DIS
LIN {X -76.4118,Y 102.7099,Z 145,A 122.3344,B 23.6846,C -1.3955,E1 23.6297,E2 684.4722} C_DIS
LIN {X -73.341,Y 104.925,Z 145,A 120.7482,B 23.6841,C -1.4036,E1 23.6333,E2 686.0438} C_DIS
LIN {X -70.69,Y 106.7292,Z 145,A 119.4807,B 23.6835,C -1.4138,E1 23.6362,E2 687.2904} C_DIS
LIN {X -66.9266,Y 109.128,Z 145,A 117.5711,B 23.6831,C -1.4214,E1 23.6407,E2 689.1873} C_DIS
LIN {X -63.4047,Y 111.2112,Z 145,A 115.675,B 23.6831,C -1.4218,E1 23.6453,E2 691.0883} C_DIS
LIN {X -59.8162,Y 113.1801,Z 145,A 113.9259,B 23.6827,C -1.4287,E1 23.6496,E2 692.8256} C_DIS
LIN {X -56.8409,Y 114.7029,Z 145,A 112.4234,B 23.6826,C -1.4308,E1 23.6533,E2 694.327} C_DIS
LIN {X -53.9777,Y 116.0779,Z 145,A 111.2274,B 23.6819,C -1.4431,E1 23.6563,E2 695.4956} C_DIS
LIN {X -51.9375,Y 117.0053,Z 145,A 109.9092,B 23.6826,C -1.4305,E1 23.6597,E2 696.8486} C_DIS
LIN {X -47.7429,Y 118.7781,Z 145,A 107.6154,B 23.6831,C -1.422,E1 23.6657,E2 699.1691} C_DIS
LIN {X -44.61,Y 119.9903,Z 145,A 106.0546,B 23.6831,C -1.4214,E1 23.6698,E2 700.7348} C_DIS
LIN {X -41.117,Y 121.2333,Z 145,A 104.8291,B 23.6819,C -1.4428,E1 23.6729,E2 701.9093} C_DIS
LIN {X -35.8566,Y 122.89,Z 145,A 102.3213,B 23.6819,C -1.4438,E1 23.6796,E2 704.4192} C_DIS
LIN {X -32.4422,Y 123.8364,Z 145,A 100.6074,B 23.6821,C -1.4397,E1 23.6843,E2 706.1463} C_DIS
LIN {X -28.4285,Y 124.8178,Z 145,A 98.8392,B 23.6817,C -1.4451,E1 23.689,E2 707.9036} C_DIS
LIN {X -24.3421,Y 125.6791,Z 145,A 96.973,B 23.6817,C -1.4467,E1 23.6941,E2 709.7679} C_DIS
LIN {X -21.0024,Y 126.2798,Z 145,A 95.443,B 23.6817,C -1.4474,E1 23.6983,E2 711.2979} C_DIS
LIN {X -17.4066,Y 126.8275,Z 145,A 93.7168,B 23.6818,C -1.4439,E1 23.7031,E2 713.0342} C_DIS
LIN {X -13.4643,Y 127.3046,Z 145,A 92.2462,B 23.6809,C -1.4589,E1 23.7071,E2 714.4684} C_DIS
LIN {X -8.1444,Y 127.7555,Z 145,A 89.6946,B 23.6813,C -1.4525,E1 23.7143,E2 717.0372} C_DIS
LIN {X -2.2155,Y 127.9955,Z 145,A 86.9873,B 23.6814,C -1.4509,E1 23.7219,E2 719.7489} C_DIS
LIN {X 5.026,Y 127.9159,Z 145,A 84.0388,B 23.6806,C -1.4649,E1 23.73,E2 722.6623} C_DIS
LIN {X 9.9892,Y 127.6259,Z 145,A 81.4401,B 23.6816,C -1.4474,E1 23.7373,E2 725.3032} C_DIS
LIN {X 13.4051,Y 127.311,Z 145,A 79.6069,B 23.6824,C -1.4335,E1 23.7425,E2 727.1699} C_DIS
LIN {X 17.0552,Y 126.8739,Z 145,A 78.1477,B 23.6819,C -1.4417,E1 23.7465,E2 728.6074} C_DIS
LIN {X 21.3756,Y 126.2175,Z 145,A 76.3587,B 23.6815,C -1.4488,E1 23.7514,E2 730.3769} C_DIS
LIN {X 25.2633,Y 125.497,Z 145,A 74.6126,B 23.6815,C -1.4491,E1 23.7562,E2 732.1199} C_DIS
LIN {X 28.6897,Y 124.7581,Z 145,A 73.0388,B 23.6815,C -1.4481,E1 23.7604,E2 733.6941} C_DIS
LIN {X 32.7373,Y 123.7578,Z 145,A 71.1934,B 23.6815,C -1.4479,E1 23.7654,E2 735.5371} C_DIS
LIN {X 36.0709,Y 122.8273,Z 145,A 69.6837,B 23.6815,C -1.4486,E1 23.7695,E2 737.0422} C_DIS
LIN {X 41.6812,Y 121.0387,Z 145,A 67.0119,B 23.6818,C -1.4447,E1 23.7766,E2 739.7184} C_DIS
LIN {X 45.6146,Y 119.614,Z 145,A 64.8432,B 23.6827,C -1.4289,E1 23.7823,E2 741.9215} C_DIS
LIN {X 48.6385,Y 118.4165,Z 145,A 63.5623,B 23.6823,C -1.4356,E1 23.7856,E2 743.1825} C_DIS
LIN {X 52.2313,Y 116.8739,Z 145,A 61.9787,B 23.6819,C -1.4416,E1 23.7896,E2 744.7473} C_DIS
LIN {X 55.0446,Y 115.5756,Z 145,A 60.5976,B 23.682,C -1.4401,E1 23.7931,E2 746.1281} C_DIS
LIN {X 57.8984,Y 114.1727,Z 145,A 59.1894,B 23.682,C -1.439,E1 23.7966,E2 747.5351} C_DIS
LIN {X 61.0173,Y 112.5392,Z 145,A 57.5737,B 23.6823,C -1.4349,E1 23.8006,E2 749.156} C_DIS
LIN {X 64.9676,Y 110.3056,Z 145,A 55.2148,B 23.6834,C -1.4163,E1 23.8064,E2 751.5536} C_DIS
LIN {X 67.9131,Y 108.5173,Z 145,A 53.9358,B 23.6828,C -1.4265,E1 23.8094,E2 752.803} C_DIS
LIN {X 70.4362,Y 106.8963,Z 145,A 52.3624,B 23.6836,C -1.4132,E1 23.8131,E2 754.4038} C_DIS
LIN {X 73.1794,Y 105.0375,Z 145,A 51.134,B 23.683,C -1.4229,E1 23.8159,E2 755.6037} C_DIS
LIN {X 76.7799,Y 102.4358,Z 145,A 49.126,B 23.6833,C -1.4184,E1 23.8204,E2 757.6152} C_DIS
LIN {X 80.08,Y 99.877,Z 145,A 47.3469,B 23.6833,C -1.4193,E1 23.8243,E2 759.3852} C_DIS
LIN {X 83.1307,Y 97.3522,Z 145,A 45.5373,B 23.6835,C -1.4141,E1 23.8282,E2 761.2004} C_DIS
LIN {X 86.3073,Y 94.5477,Z 145,A 43.6067,B 23.6838,C -1.4086,E1 23.8322,E2 763.1364} C_DIS
LIN {X 89.3908,Y 91.6378,Z 145,A 41.6929,B 23.6841,C -1.4038,E1 23.836,E2 765.0537} C_DIS
LIN {X 91.5358,Y 89.4948,Z 145,A 40.2226,B 23.6846,C -1.3953,E1 23.8389,E2 766.5384} C_DIS
LIN {X 95.1277,Y 85.6675,Z 145,A 38.0094,B 23.6845,C -1.3966,E1 23.8431,E2 768.738} C_DIS
LIN {X 98.0368,Y 82.3217,Z 145,A 36.3158,B 23.684,C -1.4062,E1 23.8461,E2 770.3997} C_DIS
LIN {X 100.6546,Y 79.0995,Z 145,A 34.2115,B 23.6849,C -1.3896,E1 23.8499,E2 772.5346} C_DIS
LIN {X 103.3178,Y 75.5882,Z 145,A 32.2662,B 23.6851,C -1.386,E1 23.8531,E2 774.4789} C_DIS
LIN {X 105.7507,Y 72.1457,Z 145,A 30.3544,B 23.6854,C -1.38,E1 23.8562,E2 776.3958} C_DIS
LIN {X 108.1216,Y 68.541,Z 145,A 28.2215,B 23.6862,C -1.365,E1 23.8594,E2 778.5544} C_DIS
LIN {X 109.886,Y 65.6747,Z 145,A 26.611,B 23.6867,C -1.3558,E1 23.8617,E2 780.1789} C_DIS
LIN {X 111.8631,Y 62.248,Z 145,A 25.2014,B 23.686,C -1.3687,E1 23.8636,E2 781.5487} C_DIS
LIN {X 113.9266,Y 58.3819,Z 145,A 23.3286,B 23.686,C -1.3677,E1 23.866,E2 783.4137} C_DIS
LIN {X 115.3484,Y 55.5201,Z 145,A 21.9605,B 23.6861,C -1.3667,E1 23.8677,E2 784.7764} C_DIS
LIN {X 116.719,Y 52.5776,Z 145,A 20.5536,B 23.6862,C -1.3648,E1 23.8693,E2 786.1799} C_DIS
LIN {X 119.4703,Y 45.9852,Z 145,A 17.1813,B 23.6872,C -1.3467,E1 23.8729,E2 789.5773} C_DIS
LIN {X 120.9024,Y 42.0743,Z 145,A 15.0238,B 23.6883,C -1.3265,E1 23.875,E2 791.7718} C_DIS
LIN {X 122.1553,Y 38.291,Z 145,A 13.5493,B 23.6878,C -1.3364,E1 23.8762,E2 793.2129} C_DIS
LIN {X 123.2728,Y 34.5177,Z 145,A 11.9662,B 23.6876,C -1.3399,E1 23.8774,E2 794.7778} C_DIS
LIN {X 124.0871,Y 31.465,Z 145,A 10.5376,B 23.6878,C -1.3348,E1 23.8784,E2 796.2103} C_DIS
LIN {X 124.939,Y 27.8982,Z 145,A 8.7705,B 23.6885,C -1.3234,E1 23.8795,E2 797.9948} C_DIS
LIN {X 125.7804,Y 23.8119,Z 145,A 7.0145,B 23.6885,C -1.3231,E1 23.8805,E2 799.7407} C_DIS
LIN {X 126.4121,Y 20.2003,Z 145,A 5.3587,B 23.6888,C -1.3171,E1 23.8812,E2 801.401} C_DIS
LIN {X 127.0208,Y 15.9337,Z 145,A 3.4043,B 23.6892,C -1.3096,E1 23.882,E2 803.3615} C_DIS
LIN {X 127.3709,Y 12.8343,Z 145,A 1.5099,B 23.6907,C -1.2803,E1 23.8825,E2 805.3166} C_DIS
LIN {X 127.754,Y 8.1684,Z 145,A 0.2541,B 23.6889,C -1.3155,E1 23.8828,E2 806.4775} C_DIS
LIN {X 128.0077,Y 1.4802,Z 145,A -2.7611,B 23.6894,C -1.3047,E1 23.8831,E2 809.5004} C_DIS
LIN {X 127.9373,Y -4.4772,Z 145,A -6.1116,B 23.6916,C -1.2617,E1 23.8828,E2 812.936} C_DIS
LIN {X 127.7125,Y -8.8034,Z 145,A -7.5948,B 23.6908,C -1.2782,E1 23.8826,E2 814.3691} C_DIS
LIN {X 127.3961,Y -12.5723,Z 145,A -9.5728,B 23.6918,C -1.2584,E1 23.8821,E2 816.3836} C_DIS
LIN {X 126.9934,Y -16.1381,Z 145,A -10.9931,B 23.6916,C -1.2625,E1 23.8816,E2 817.7851} C_DIS
LIN {X 126.3191,Y -20.7667,Z 145,A -12.8959,B 23.6914,C -1.2652,E1 23.8808,E2 819.6691} C_DIS
LIN {X 125.7275,Y -24.0891,Z 145,A -14.3263,B 23.6914,C -1.2644,E1 23.88,E2 821.0928} C_DIS
LIN {X 125.0793,Y -27.2561,Z 145,A -15.8448,B 23.6919,C -1.2561,E1 23.8792,E2 822.6223} C_DIS
LIN {X 124.1226,Y -31.3252,Z 145,A -17.6557,B 23.6921,C -1.2531,E1 23.878,E2 824.4296} C_DIS
LIN {X 123.2568,Y -34.5749,Z 145,A -18.9873,B 23.6919,C -1.257,E1 23.877,E2 825.7433} C_DIS
LIN {X 122.1043,Y -38.4505,Z 145,A -20.8241,B 23.6922,C -1.2499,E1 23.8755,E2 827.5867} C_DIS
LIN {X 121.4602,Y -40.4358,Z 145,A -22.6509,B 23.6945,C -1.2024,E1 23.8738,E2 829.5201} C_DIS
LIN {X 119.5583,Y -45.7588,Z 145,A -24.32,B 23.6928,C -1.2374,E1 23.8723,E2 831.0927} C_DIS
LIN {X 116.132,Y -53.8607,Z 145,A -28.2694,B 23.6935,C -1.2246,E1 23.8679,E2 835.0508} C_DIS
LIN {X 114.8708,Y -56.5005,Z 145,A -29.5505,B 23.6935,C -1.222,E1 23.8663,E2 836.3309} C_DIS
LIN {X 113.4092,Y -59.3798,Z 145,A -31.0194,B 23.6938,C -1.2165,E1 23.8645,E2 837.8052} C_DIS
LIN {X 111.5541,Y -62.7996,Z 145,A -32.8365,B 23.6943,C -1.2076,E1 23.862,E2 839.6344} C_DIS
LIN {X 109.5293,Y -66.2679,Z 145,A -35.2463,B 23.696,C -1.1719,E1 23.8584,E2 842.1194} C_DIS
LIN {X 106.7537,Y -70.6528,Z 145,A -36.8193,B 23.6945,C -1.2025,E1 23.8562,E2 843.6083} C_DIS
LIN {X 103.4489,Y -75.4091,Z 145,A -39.5545,B 23.6952,C -1.1882,E1 23.8517,E2 846.3648} C_DIS
LIN {X 101.4864,Y -78.0301,Z 145,A -41.4144,B 23.6963,C -1.1646,E1 23.8485,E2 848.2736} C_DIS
LIN {X 98.8076,Y -81.3956,Z 145,A -43.0715,B 23.6959,C -1.1728,E1 23.8456,E2 849.9025} C_DIS
LIN {X 95.6666,Y -85.0654,Z 145,A -45.0717,B 23.6959,C -1.1752,E1 23.8419,E2 851.8872} C_DIS
LIN {X 92.4989,Y -88.4988,Z 145,A -47.252,B 23.6963,C -1.1655,E1 23.8377,E2 854.0814} C_DIS
LIN {X 88.2434,Y -92.743,Z 145,A -49.7662,B 23.6962,C -1.1676,E1 23.8328,E2 856.5791} C_DIS
LIN {X 85.102,Y -95.6341,Z 145,A -51.7435,B 23.6965,C -1.1598,E1 23.8286,E2 858.5672} C_DIS
LIN {X 82.9513,Y -97.5047,Z 145,A -53.0808,B 23.6968,C -1.1539,E1 23.8258,E2 859.9137} C_DIS
LIN {X 77.7414,Y -101.7072,Z 145,A -55.9462,B 23.6968,C -1.1538,E1 23.8195,E2 862.7681} C_DIS
LIN {X 74.1656,Y -104.344,Z 145,A -57.8515,B 23.6968,C -1.1537,E1 23.8152,E2 864.6665} C_DIS
LIN {X 70.837,Y -106.6316,Z 145,A -59.4443,B 23.6965,C -1.1606,E1 23.8116,E2 866.2363} C_DIS
LIN {X 67.8744,Y -108.5414,Z 145,A -61.3306,B 23.6973,C -1.1424,E1 23.8071,E2 868.1613} C_DIS
LIN {X 64.4326,Y -110.6194,Z 145,A -63.407,B 23.6981,C -1.1256,E1 23.802,E2 870.2727} C_DIS
LIN {X 61.2459,Y -112.4144,Z 145,A -64.9948,B 23.6981,C -1.1251,E1 23.7981,E2 871.8568} C_DIS
LIN {X 58.2715,Y -113.9828,Z 145,A -66.1462,B 23.6974,C -1.1398,E1 23.7954,E2 872.9684} C_DIS
LIN {X 55.1614,Y -115.5198,Z 145,A -67.6027,B 23.6974,C -1.142,E1 23.7917,E2 874.4155} C_DIS
LIN {X 52.9241,Y -116.564,Z 145,A -69.6382,B 23.6994,C -1.0953,E1 23.7863,E2 876.5615} C_DIS
LIN {X 47.4927,Y -118.879,Z 145,A -71.5437,B 23.698,C -1.1269,E1 23.7816,E2 878.3837} C_DIS
LIN {X 43.6616,Y -120.3385,Z 145,A -73.0136,B 23.6973,C -1.1422,E1 23.7778,E2 879.8125} C_DIS
LIN {X 37.7514,Y -122.3215,Z 145,A -76.0969,B 23.6981,C -1.1245,E1 23.7696,E2 882.9335} C_DIS
LIN {X 33.994,Y -123.4192,Z 145,A -77.8944,B 23.6983,C -1.1204,E1 23.7647,E2 884.738} C_DIS
LIN {X 30.0582,Y -124.4354,Z 145,A -79.5841,B 23.6981,C -1.1248,E1 23.7602,E2 886.4141} C_DIS
LIN {X 26.5582,Y -125.23,Z 145,A -81.287,B 23.6984,C -1.1187,E1 23.7555,E2 888.1298} C_DIS
LIN {X 22.754,Y -125.9761,Z 145,A -82.946,B 23.6983,C -1.1209,E1 23.7509,E2 889.7813} C_DIS
LIN {X 15.7641,Y -127.0416,Z 145,A -86.1651,B 23.6985,C -1.1161,E1 23.742,E2 893.0092} C_DIS
LIN {X 11.0546,Y -127.5366,Z 145,A -87.9804,B 23.6979,C -1.1294,E1 23.7371,E2 894.79} C_DIS
LIN {X 6.0201,Y -127.8736,Z 145,A -90.5918,B 23.6987,C -1.1117,E1 23.7297,E2 897.4445} C_DIS
LIN {X 0.9107,Y -127.9787,Z 145,A -92.4381,B 23.6978,C -1.1324,E1 23.7247,E2 899.2388} C_DIS
Enddeposition()
LIN {X 0.9107,Y -127.9787,Z 145,A -92.4381,B 23.6978,C -1.1324,E1 23.7247,E2 899.2388} C_DIS
Startdeposition()
$VEL.CP = VEL_PRINT
LIN {X 3.7604,Y -126.9989,Z 145,A -90.5632,B 22.884,C -1.0204,E1 22.9117,E2 897.543} C_DIS
LIN {X 9.8324,Y -126.6746,Z 145,A -87.7254,B 22.8838,C -1.0259,E1 22.9196,E2 894.6923} C_DIS
LIN {X 14.235,Y -126.2559,Z 145,A -85.8676,B 22.884,C -1.0207,E1 22.9247,E2 892.8493} C_DIS
LIN {X 17.8955,Y -125.7876,Z 145,A -83.9194,B 22.8834,C -1.0349,E1 22.9302,E2 890.8663} C_DIS
LIN {X 22.3494,Y -125.073,Z 145,A -82.0867,B 22.8838,C -1.0271,E1 22.9352,E2 889.0558} C_DIS
LIN {X 26.2888,Y -124.3058,Z 145,A -80.2414,B 22.8836,C -1.0303,E1 22.9403,E2 887.2048} C_DIS
LIN {X 29.8375,Y -123.5009,Z 145,A -78.6707,B 22.8836,C -1.0286,E1 22.9445,E2 885.6409} C_DIS
LIN {X 33.7084,Y -122.502,Z 145,A -76.8041,B 22.8835,C -1.0334,E1 22.9496,E2 883.7652} C_DIS
LIN {X 37.1497,Y -121.5015,Z 145,A -75.4502,B 22.8839,C -1.023,E1 22.9531,E2 882.4406} C_DIS
LIN {X 45.2567,Y -118.7227,Z 145,A -71.4658,B 22.8835,C -1.0333,E1 22.9637,E2 878.4385} C_DIS
LIN {X 53.4321,Y -115.2723,Z 145,A -67.4293,B 22.8832,C -1.0407,E1 22.9741,E2 874.3937} C_DIS
LIN {X 56.5751,Y -113.7633,Z 145,A -65.7264,B 22.8828,C -1.0494,E1 22.9784,E2 872.6735} C_DIS
LIN {X 62.6564,Y -110.5326,Z 145,A -62.6332,B 22.8826,C -1.0542,E1 22.986,E2 869.578} C_DIS
LIN {X 66.4125,Y -108.3168,Z 145,A -60.762,B 22.8826,C -1.0533,E1 22.9904,E2 867.7155} C_DIS
LIN {X 69.6125,Y -106.289,Z 145,A -58.9931,B 22.8824,C -1.0594,E1 22.9946,E2 865.9371} C_DIS
LIN {X 74.3071,Y -103.0617,Z 145,A -56.4607,B 22.8822,C -1.0629,E1 23.0004,E2 863.4056} C_DIS
LIN {X 80.4191,Y -98.3663,Z 145,A -52.5531,B 22.881,C -1.0912,E1 23.0091,E2 859.4415} C_DIS
LIN {X 83.7648,Y -95.5338,Z 145,A -51.0196,B 22.8817,C -1.0743,E1 23.0122,E2 857.958} C_DIS
LIN {X 86.8795,Y -92.7107,Z 145,A -48.7353,B 22.8807,C -1.0975,E1 23.017,E2 855.6245} C_DIS
LIN {X 89.8843,Y -89.8002,Z 145,A -46.8101,B 22.8804,C -1.104,E1 23.0208,E2 853.6918} C_DIS
LIN {X 92.9459,Y -86.6269,Z 145,A -45.3174,B 22.8812,C -1.0849,E1 23.0235,E2 852.2551} C_DIS
LIN {X 95.417,Y -83.898,Z 145,A -43.1855,B 22.88,C -1.112,E1 23.0276,E2 850.0643} C_DIS
LIN {X 98.2663,Y -80.5414,Z 145,A -40.868,B 22.879,C -1.1335,E1 23.0317,E2 847.7036} C_DIS
LIN {X 102.0438,Y -75.6985,Z 145,A -39.2081,B 22.8811,C -1.0869,E1 23.0343,E2 846.1717} C_DIS
LIN {X 105.5193,Y -70.7736,Z 145,A -36.2178,B 22.8802,C -1.1075,E1 23.0392,E2 843.1448} C_DIS
LIN {X 108.582,Y -65.9787,Z 145,A -33.669,B 22.8799,C -1.114,E1 23.0429,E2 840.5937} C_DIS
LIN {X 110.7375,Y -62.2926,Z 145,A -31.7188,B 22.8796,C -1.1208,E1 23.0457,E2 838.6373} C_DIS
LIN {X 112.9848,Y -58.1154,Z 145,A -29.6482,B 22.8795,C -1.1238,E1 23.0483,E2 836.5711} C_DIS
LIN {X 114.5631,Y -54.9365,Z 145,A -28.1664,B 22.8795,C -1.1228,E1 23.0501,E2 835.1005} C_DIS
LIN {X 117.9372,Y -47.2606,Z 145,A -24.3159,B 22.8788,C -1.1376,E1 23.0544,E2 831.2354} C_DIS
LIN {X 119.5463,Y -43.0279,Z 145,A -21.9339,B 22.8777,C -1.1606,E1 23.0568,E2 828.8094} C_DIS
LIN {X 120.807,Y -39.3562,Z 145,A -20.6539,B 22.8786,C -1.143,E1 23.0578,E2 827.5823} C_DIS
LIN {X 121.7731,Y -36.2542,Z 145,A -18.9811,B 22.8779,C -1.1577,E1 23.0592,E2 825.8823} C_DIS
LIN {X 123.0566,Y -31.6219,Z 145,A -16.9513,B 22.8779,C -1.1579,E1 23.0607,E2 823.8651} C_DIS
LIN {X 123.8409,Y -28.3934,Z 145,A -15.5591,B 22.8779,C -1.1575,E1 23.0615,E2 822.4828} C_DIS
LIN {X 124.4708,Y -25.4911,Z 145,A -14.1747,B 22.8776,C -1.164,E1 23.0623,E2 821.0907} C_DIS
LIN {X 125.1495,Y -21.9222,Z 145,A -12.454,B 22.8771,C -1.1732,E1 23.0632,E2 819.3574} C_DIS
LIN {X 125.7714,Y -18.0088,Z 145,A -10.2164,B 22.8757,C -1.2011,E1 23.0641,E2 817.0631} C_DIS
LIN {X 126.333,Y -13.5191,Z 145,A -8.7548,B 22.8768,C -1.1793,E1 23.0646,E2 815.6667} C_DIS
LIN {X 126.6848,Y -9.6933,Z 145,A -7.0434,B 22.8766,C -1.1839,E1 23.065,E2 813.9549} C_DIS
LIN {X 126.8839,Y -6.5823,Z 145,A -5.4163,B 22.8758,C -1.1992,E1 23.0652,E2 812.2992} C_DIS
LIN {X 127.0571,Y 0.1112,Z 145,A -2.54,B 22.8757,C -1.2019,E1 23.0653,E2 809.4349} C_DIS
LIN {X 127.0157,Y 3.1572,Z 145,A -0.8584,B 22.8747,C -1.2214,E1 23.0653,E2 807.7144} C_DIS
LIN {X 126.8616,Y 7.0261,Z 145,A 0.5177,B 22.8754,C -1.2089,E1 23.065,E2 806.3794} C_DIS
LIN {X 126.4767,Y 12.1009,Z 145,A 2.7685,B 22.8751,C -1.2141,E1 23.0645,E2 804.13} C_DIS
LIN {X 126.0047,Y 16.2983,Z 145,A 4.5297,B 22.8751,C -1.2132,E1 23.0639,E2 802.3826} C_DIS
LIN {X 125.5368,Y 19.578,Z 145,A 6.1124,B 22.8747,C -1.2222,E1 23.0633,E2 800.7871} C_DIS
LIN {X 124.8702,Y 23.4594,Z 145,A 7.9259,B 22.8743,C -1.2296,E1 23.0624,E2 798.9664} C_DIS
LIN {X 124.0889,Y 27.2934,Z 145,A 9.716,B 22.874,C -1.2364,E1 23.0613,E2 797.1706} C_DIS
LIN {X 123.1925,Y 31.0863,Z 145,A 11.3601,B 22.874,C -1.2364,E1 23.0602,E2 795.5371} C_DIS
LIN {X 122.3551,Y 34.234,Z 145,A 12.7914,B 22.8738,C -1.239,E1 23.0592,E2 794.1081} C_DIS
LIN {X 121.4396,Y 37.3521,Z 145,A 14.0666,B 22.8741,C -1.2342,E1 23.0582,E2 792.853} C_DIS
LIN {X 119.4595,Y 43.2685,Z 145,A 16.7862,B 22.8739,C -1.2381,E1 23.0558,E2 790.1405} C_DIS
LIN {X 116.3646,Y 51.0136,Z 145,A 20.9162,B 22.8724,C -1.2666,E1 23.0514,E2 785.9626} C_DIS
LIN {X 114.7038,Y 54.6419,Z 145,A 22.596,B 22.8724,C -1.266,E1 23.0494,E2 784.2945} C_DIS
LIN {X 113.2487,Y 57.597,Z 145,A 24.0336,B 22.8724,C -1.2679,E1 23.0476,E2 782.8606} C_DIS
LIN {X 111.6405,Y 60.6598,Z 145,A 25.5427,B 22.8722,C -1.2697,E1 23.0456,E2 781.3556} C_DIS
LIN {X 109.4574,Y 64.5156,Z 145,A 27.607,B 22.8718,C -1.2782,E1 23.0428,E2 779.2811} C_DIS
LIN {X 107.0526,Y 68.4318,Z 145,A 29.7619,B 22.8713,C -1.2877,E1 23.0396,E2 777.1141} C_DIS
LIN {X 104.5476,Y 72.2017,Z 145,A 31.76,B 22.8711,C -1.2908,E1 23.0364,E2 775.1188} C_DIS
LIN {X 102.1288,Y 75.5844,Z 145,A 33.6621,B 22.8708,C -1.2968,E1 23.0333,E2 773.2116} C_DIS
LIN {X 100.4134,Y 77.848,Z 145,A 35.0984,B 22.8702,C -1.3074,E1 23.0308,E2 771.7558} C_DIS
LIN {X 97.0792,Y 81.9692,Z 145,A 37.342,B 22.8703,C -1.306,E1 23.0268,E2 769.5271} C_DIS
LIN {X 93.8062,Y 85.6955,Z 145,A 39.775,B 22.8695,C -1.3204,E1 23.0223,E2 767.0691} C_DIS
LIN {X 91.5194,Y 88.1333,Z 145,A 41.0456,B 22.8699,C -1.3125,E1 23.0198,E2 765.8249} C_DIS
LIN {X 88.5835,Y 91.0835,Z 145,A 42.9059,B 22.8698,C -1.3157,E1 23.0161,E2 763.965} C_DIS
LIN {X 85.3899,Y 94.0836,Z 145,A 44.8634,B 22.8696,C -1.3189,E1 23.0121,E2 762.0081} C_DIS
LIN {X 82.1036,Y 96.965,Z 145,A 46.8313,B 22.8694,C -1.3226,E1 23.008,E2 760.0392} C_DIS
LIN {X 78.8512,Y 99.6281,Z 145,A 48.6463,B 22.8694,C -1.3224,E1 23.004,E2 758.2323} C_DIS
LIN {X 75.5746,Y 102.1361,Z 145,A 50.605,B 22.869,C -1.3303,E1 22.9996,E2 756.2611} C_DIS
LIN {X 70.9578,Y 105.3957,Z 145,A 53.157,B 22.8687,C -1.3348,E1 22.9938,E2 753.7073} C_DIS
LIN {X 67.23,Y 107.8114,Z 145,A 54.848,B 22.8694,C -1.3234,E1 22.9899,E2 752.0515} C_DIS
LIN {X 63.9704,Y 109.7774,Z 145,A 56.5736,B 22.8692,C -1.3264,E1 22.9857,E2 750.3242} C_DIS
LIN {X 60.9214,Y 111.4978,Z 145,A 58.387,B 22.8685,C -1.3395,E1 22.9812,E2 748.483} C_DIS
LIN {X 57.7213,Y 113.1854,Z 145,A 59.9121,B 22.8686,C -1.3367,E1 22.9775,E2 746.9696} C_DIS
LIN {X 55.0418,Y 114.5127,Z 145,A 61.2264,B 22.8686,C -1.3368,E1 22.9742,E2 745.6589} C_DIS
LIN {X 52.2803,Y 115.8,Z 145,A 62.6607,B 22.8684,C -1.3412,E1 22.9705,E2 744.2173} C_DIS
LIN {X 49.3061,Y 117.0971,Z 145,A 64.1284,B 22.8683,C -1.3431,E1 22.9668,E2 742.7488} C_DIS
LIN {X 46.6934,Y 118.1648,Z 145,A 66.062,B 22.8665,C -1.3749,E1 22.9616,E2 740.7382} C_DIS
LIN {X 41.948,Y 119.9299,Z 145,A 68.2735,B 22.8665,C -1.3736,E1 22.9557,E2 738.5348} C_DIS
LIN {X 37.3974,Y 121.4257,Z 145,A 69.8165,B 22.8681,C -1.3469,E1 22.9518,E2 737.0635} C_DIS
LIN {X 34.0727,Y 122.4002,Z 145,A 71.3912,B 22.868,C -1.3486,E1 22.9476,E2 735.4875} C_DIS
LIN {X 30.023,Y 123.4561,Z 145,A 73.233,B 22.868,C -1.3477,E1 22.9426,E2 733.651} C_DIS
LIN {X 26.7387,Y 124.2087,Z 145,A 74.8047,B 22.8678,C -1.3509,E1 22.9383,E2 732.0734} C_DIS
LIN {X 22.686,Y 125.0128,Z 145,A 76.6556,B 22.8678,C -1.3511,E1 22.9332,E2 730.2243} C_DIS
LIN {X 19.1673,Y 125.6004,Z 145,A 78.1829,B 22.868,C -1.348,E1 22.9291,E2 728.7068} C_DIS
LIN {X 13.7051,Y 126.313,Z 145,A 80.7203,B 22.8678,C -1.3509,E1 22.922,E2 726.164} C_DIS
LIN {X 9.7761,Y 126.6787,Z 145,A 82.3878,B 22.8681,C -1.346,E1 22.9174,E2 724.5101} C_DIS
LIN {X 5.4441,Y 126.9386,Z 145,A 84.4773,B 22.8678,C -1.352,E1 22.9115,E2 722.4062} C_DIS
LIN {X -0.0954,Y 127.0558,Z 145,A 87.0597,B 22.8676,C -1.3553,E1 22.9043,E2 719.8154} C_DIS
LIN {X -4.0584,Y 126.9906,Z 145,A 88.8701,B 22.8676,C -1.3559,E1 22.8992,E2 718.0033} C_DIS
LIN {X -9.2463,Y 126.7174,Z 145,A 91.4258,B 22.8671,C -1.3645,E1 22.8921,E2 715.4244} C_DIS
LIN {X -12.6904,Y 126.4201,Z 145,A 92.7783,B 22.8676,C -1.3546,E1 22.8884,E2 714.0968} C_DIS
LIN {X -16.6024,Y 125.9648,Z 145,A 94.3333,B 22.8682,C -1.3438,E1 22.8841,E2 712.5683} C_DIS
LIN {X -19.9588,Y 125.4778,Z 145,A 96.078,B 22.8678,C -1.3523,E1 22.8793,E2 710.8002} C_DIS
LIN {X -23.8647,Y 124.7927,Z 145,A 97.7478,B 22.8681,C -1.3457,E1 22.8747,E2 709.1453} C_DIS
LIN {X -27.5213,Y 124.0397,Z 145,A 99.5392,B 22.8679,C -1.349,E1 22.8698,E2 707.343} C_DIS
LIN {X -30.7938,Y 123.2668,Z 145,A 101.0041,B 22.8681,C -1.3454,E1 22.8658,E2 705.8853} C_DIS
LIN {X -34.1845,Y 122.3689,Z 145,A 102.4677,B 22.8685,C -1.3386,E1 22.8619,E2 704.4366} C_DIS
LIN {X -41.0126,Y 120.2542,Z 145,A 105.6896,B 22.8687,C -1.3348,E1 22.8534,E2 701.2183} C_DIS
LIN {X -47.0798,Y 118.0101,Z 145,A 108.6853,B 22.8687,C -1.3344,E1 22.8455,E2 698.2169} C_DIS
LIN {X -50.022,Y 116.7933,Z 145,A 110.196,B 22.8687,C -1.3356,E1 22.8416,E2 696.6992} C_DIS
LIN {X -52.8131,Y 115.5585,Z 145,A 111.5479,B 22.8689,C -1.3325,E1 22.8382,E2 695.3517} C_DIS
LIN {X -55.986,Y 114.0539,Z 145,A 113.1097,B 22.869,C -1.3291,E1 22.8343,E2 693.7941} C_DIS
LIN {X -58.9962,Y 112.5261,Z 145,A 114.6148,B 22.8692,C -1.3258,E1 22.8305,E2 692.2928} C_DIS
LIN {X -62.6413,Y 110.5412,Z 145,A 116.6184,B 22.8691,C -1.3283,E1 22.8256,E2 690.2767} C_DIS
LIN {X -66.2375,Y 108.4242,Z 145,A 118.501,B 22.8693,C -1.3249,E1 22.8211,E2 688.3964} C_DIS
LIN {X -69.971,Y 106.053,Z 145,A 120.4092,B 22.8697,C -1.3174,E1 22.8167,E2 686.5007} C_DIS
LIN {X -75.1291,Y 102.4636,Z 145,A 123.2986,B 22.8699,C -1.3141,E1 22.8101,E2 683.6089} C_DIS
LIN {X -78.3204,Y 100.0456,Z 145,A 125.1739,B 22.8699,C -1.3133,E1 22.8059,E2 681.7282} C_DIS
LIN {X -80.9643,Y 97.918,Z 145,A 126.8209,B 22.8699,C -1.3149,E1 22.8023,E2 680.0701} C_DIS
LIN {X -85.8956,Y 93.6222,Z 145,A 129.6726,B 22.8704,C -1.304,E1 22.7964,E2 677.234} C_DIS
LIN {X -89.1796,Y 90.5,Z 145,A 131.6057,B 22.8709,C -1.2945,E1 22.7926,E2 675.3166} C_DIS
LIN {X -92.0151,Y 87.6151,Z 145,A 133.8927,B 22.8701,C -1.3097,E1 22.788,E2 672.9795} C_DIS
LIN {X -94.5867,Y 84.8323,Z 145,A 135.2756,B 22.8711,C -1.2916,E1 22.7855,E2 671.6366} C_DIS
LIN {X -97.5594,Y 81.3968,Z 145,A 137.1242,B 22.8718,C -1.2779,E1 22.7822,E2 669.814} C_DIS
LIN {X -99.3183,Y 79.2405,Z 145,A 138.9677,B 22.8707,C -1.2994,E1 22.7789,E2 667.9053} C_DIS
LIN {X -101.7461,Y 76.0983,Z 145,A 140.3984,B 22.8717,C -1.2794,E1 22.7766,E2 666.5189} C_DIS
LIN {X -104.2694,Y 72.602,Z 145,A 142.3721,B 22.8719,C -1.2754,E1 22.7734,E2 664.5449} C_DIS
LIN {X -106.7494,Y 68.9046,Z 145,A 144.4021,B 22.8722,C -1.2707,E1 22.7703,E2 662.5158} C_DIS
LIN {X -108.9095,Y 65.437,Z 145,A 146.2238,B 22.8725,C -1.2646,E1 22.7676,E2 660.6996} C_DIS
LIN {X -110.9365,Y 61.9386,Z 145,A 148.046,B 22.8728,C -1.2593,E1 22.7651,E2 658.8806} C_DIS
LIN {X -113.0829,Y 57.9225,Z 145,A 150.0572,B 22.8732,C -1.2515,E1 22.7625,E2 656.8777} C_DIS
LIN {X -114.5584,Y 54.9463,Z 145,A 151.3039,B 22.874,C -1.2366,E1 22.761,E2 655.6621} C_DIS
LIN {X -116.5105,Y 50.676,Z 145,A 153.9203,B 22.8732,C -1.251,E1 22.758,E2 652.9926} C_DIS
LIN {X -118.3887,Y 46.1173,Z 145,A 155.9239,B 22.874,C -1.235,E1 22.7559,E2 651.018} C_DIS
LIN {X -119.4725,Y 43.2326,Z 145,A 157.5385,B 22.8738,C -1.2401,E1 22.7544,E2 649.3802} C_DIS
LIN {X -121.0921,Y 38.4639,Z 145,A 160.2208,B 22.8732,C -1.2503,E1 22.752,E2 646.6546} C_DIS
LIN {X -122.4303,Y 33.9649,Z 145,A 161.8105,B 22.8747,C -1.2215,E1 22.7509,E2 645.1292} C_DIS
LIN {X -123.3168,Y 30.5968,Z 145,A 163.8449,B 22.874,C -1.2359,E1 22.7495,E2 643.0444} C_DIS
LIN {X -124.2487,Y 26.5534,Z 145,A 165.3323,B 22.8751,C -1.2139,E1 22.7486,E2 641.6043} C_DIS
LIN {X -125.0444,Y 22.5093,Z 145,A 167.0972,B 22.8756,C -1.204,E1 22.7477,E2 639.8533} C_DIS
LIN {X -125.6488,Y 18.8542,Z 145,A 168.8805,B 22.8756,C -1.2034,E1 22.7469,E2 638.0601} C_DIS
LIN {X -126.1522,Y 15.1127,Z 145,A 170.4482,B 22.8762,C -1.1923,E1 22.7464,E2 636.5107} C_DIS
LIN {X -126.5167,Y 11.6842,Z 145,A 172.1283,B 22.8762,C -1.1925,E1 22.7459,E2 634.819} C_DIS
LIN {X -126.8177,Y 7.7514,Z 145,A 173.861,B 22.8765,C -1.1848,E1 22.7456,E2 633.0946} C_DIS
LIN {X -126.9974,Y 3.8133,Z 145,A 175.658,B 22.8768,C -1.1799,E1 22.7454,E2 631.2983} C_DIS
LIN {X -127.057,Y -0.1353,Z 145,A 177.5879,B 22.8768,C -1.1803,E1 22.7454,E2 629.3545} C_DIS
LIN {X -126.9725,Y -4.5747,Z 145,A 179.4849,B 22.8773,C -1.1696,E1 22.7455,E2 627.4728} C_DIS
LIN {X -126.7909,Y -8.1854,Z 145,A -178.8046,B 22.8773,C -1.1677,E1 22.7458,E2 625.7558} C_DIS
LIN {X -126.4957,Y -11.9031,Z 145,A -177.1867,B 22.8778,C -1.1597,E1 22.7462,E2 624.148} C_DIS
LIN {X -126.0707,Y -15.7948,Z 145,A -175.3204,B 22.8778,C -1.1582,E1 22.7468,E2 622.273} C_DIS
LIN {X -125.5617,Y -19.4172,Z 145,A -173.7734,B 22.8783,C -1.1488,E1 22.7474,E2 620.7403} C_DIS
LIN {X -124.9295,Y -23.1494,Z 145,A -171.9426,B 22.8783,C -1.1486,E1 22.7483,E2 618.898} C_DIS
LIN {X -124.1963,Y -26.7961,Z 145,A -170.3627,B 22.8787,C -1.1393,E1 22.7492,E2 617.3319} C_DIS
LIN {X -123.3283,Y -30.5512,Z 145,A -168.6687,B 22.8791,C -1.1321,E1 22.7503,E2 615.6456} C_DIS
LIN {X -122.1495,Y -34.9656,Z 145,A -166.616,B 22.8794,C -1.1254,E1 22.7518,E2 613.5969} C_DIS
LIN {X -120.4543,Y -40.4174,Z 145,A -163.9357,B 22.8795,C -1.1221,E1 22.7541,E2 610.9082} C_DIS
LIN {X -119.0578,Y -44.362,Z 145,A -162.0285,B 22.8798,C -1.1174,E1 22.7559,E2 609.0013} C_DIS
LIN {X -117.7696,Y -47.6766,Z 145,A -160.4282,B 22.88,C -1.1126,E1 22.7576,E2 607.4037} C_DIS
LIN {X -116.1414,Y -51.5172,Z 145,A -158.49,B 22.8801,C -1.1095,E1 22.7597,E2 605.4614} C_DIS
LIN {X -114.9445,Y -54.138,Z 145,A -157.2844,B 22.8805,C -1.1019,E1 22.7611,E2 604.2684} C_DIS
LIN {X -113.3999,Y -57.2999,Z 145,A -155.736,B 22.8807,C -1.0958,E1 22.763,E2 602.7264} C_DIS
LIN {X -112.3499,Y -59.3318,Z 145,A -153.9122,B 22.8793,C -1.1267,E1 22.7656,E2 600.812} C_DIS
LIN {X -109.8462,Y -63.8516,Z 145,A -152.165,B 22.8808,C -1.0955,E1 22.7679,E2 599.1356} C_DIS
LIN {X -107.7429,Y -67.3401,Z 145,A -150.3395,B 22.881,C -1.0902,E1 22.7705,E2 597.3135} C_DIS
LIN {X -106.0801,Y -69.9298,Z 145,A -148.2991,B 22.8799,C -1.1145,E1 22.7738,E2 595.1987} C_DIS
LIN {X -103.1143,Y -74.2345,Z 145,A -146.8189,B 22.8819,C -1.071,E1 22.776,E2 593.8231} C_DIS
LIN {X -99.3833,Y -79.1589,Z 145,A -143.7823,B 22.8817,C -1.0749,E1 22.7812,E2 590.7606} C_DIS
LIN {X -96.6006,Y -82.5324,Z 145,A -141.7471,B 22.8817,C -1.073,E1 22.7849,E2 588.72} C_DIS
LIN {X -93.7547,Y -85.7514,Z 145,A -139.7819,B 22.8819,C -1.0698,E1 22.7886,E2 586.7534} C_DIS
LIN {X -90.6747,Y -89.0015,Z 145,A -137.8086,B 22.8822,C -1.0634,E1 22.7924,E2 584.7871} C_DIS
LIN {X -87.5458,Y -92.0815,Z 145,A -135.7792,B 22.8822,C -1.0614,E1 22.7964,E2 582.7536} C_DIS
LIN {X -84.3598,Y -95.0087,Z 145,A -133.8119,B 22.8824,C -1.0582,E1 22.8005,E2 580.7859} C_DIS
LIN {X -80.9102,Y -97.9629,Z 145,A -131.908,B 22.8829,C -1.048,E1 22.8046,E2 578.9002} C_DIS
LIN {X -77.9037,Y -100.3702,Z 145,A -130.2447,B 22.8831,C -1.0417,E1 22.8082,E2 577.2466} C_DIS
LIN {X -74.4397,Y -102.9651,Z 145,A -127.8801,B 22.8825,C -1.0563,E1 22.8136,E2 574.835} C_DIS
LIN {X -70.1612,Y -105.9278,Z 145,A -125.8465,B 22.8833,C -1.0387,E1 22.8182,E2 572.8392} C_DIS
LIN {X -66.7424,Y -108.1145,Z 145,A -123.9363,B 22.8833,C -1.0394,E1 22.8227,E2 570.9205} C_DIS
LIN {X -63.3431,Y -110.1406,Z 145,A -122.0625,B 22.8832,C -1.0407,E1 22.8273,E2 569.0371} C_DIS
LIN {X -59.6238,Y -112.1965,Z 145,A -120.1623,B 22.8833,C -1.0374,E1 22.8319,E2 567.1395} C_DIS
LIN {X -56.4825,Y -113.809,Z 145,A -118.6523,B 22.8836,C -1.0318,E1 22.8357,E2 565.6395} C_DIS
LIN {X -53.4984,Y -115.2417,Z 145,A -117.2394,B 22.8838,C -1.0265,E1 22.8392,E2 564.2363} C_DIS
LIN {X -50.007,Y -116.7998,Z 145,A -114.6861,B 22.8823,C -1.0616,E1 22.846,E2 561.5859} C_DIS
LIN {X -44.9862,Y -118.824,Z 145,A -112.4435,B 22.8828,C -1.0504,E1 22.8518,E2 559.3671} C_DIS
LIN {X -40.7863,Y -120.3314,Z 145,A -110.8781,B 22.8837,C -1.0286,E1 22.8558,E2 557.8546} C_DIS
LIN {X -37.3854,Y -121.4294,Z 145,A -109.3595,B 22.8839,C -1.0232,E1 22.8598,E2 556.3468} C_DIS
LIN {X -34.3526,Y -122.3219,Z 145,A -107.9762,B 22.884,C -1.0204,E1 22.8635,E2 554.9684} C_DIS
LIN {X -31.0846,Y -123.193,Z 145,A -106.3735,B 22.884,C -1.0229,E1 22.8679,E2 553.3567} C_DIS
LIN {X -27.0535,Y -124.1407,Z 145,A -104.5695,B 22.884,C -1.0191,E1 22.8728,E2 551.5598} C_DIS
LIN {X -24.0714,Y -124.7532,Z 145,A -103.163,B 22.884,C -1.02,E1 22.8766,E2 550.1492} C_DIS
LIN {X -20.7909,Y -125.3416,Z 145,A -101.117,B 22.883,C -1.0442,E1 22.8825,E2 548.0388} C_DIS
LIN {X -16.4703,Y -125.9822,Z 145,A -99.6412,B 22.884,C -1.0213,E1 22.8864,E2 546.6208} C_DIS
LIN {X -12.3986,Y -126.4481,Z 145,A -97.4065,B 22.8833,C -1.0387,E1 22.8927,E2 544.3399} C_DIS
LIN {X -8.4828,Y -126.7726,Z 145,A -96.1234,B 22.8842,C -1.0163,E1 22.8961,E2 543.1138} C_DIS
LIN {X -2.4103,Y -127.0319,Z 145,A -93.2955,B 22.884,C -1.0205,E1 22.9041,E2 540.2746} C_DIS
LIN {X 0.8965,Y -127.0425,Z 145,A -91.7579,B 22.884,C -1.0231,E1 22.9084,E2 538.7304} C_DIS
Enddeposition()
LIN {X 0.8965,Y -127.0425,Z 145,A -91.7579,B 22.884,C -1.0231,E1 22.9084,E2 538.7304} C_DIS
Startdeposition()
$VEL.CP = VEL_PRINT
LIN {X -0.6901,Y -126.0923,Z 145,A -93.0071,B 21.9732,C -0.8509,E1 21.9872,E2 540.3183} C_DIS
LIN {X -5.49,Y -125.9759,Z 145,A -95.0795,B 21.973,C -0.8553,E1 21.9814,E2 542.3792} C_DIS
LIN {X -8.4113,Y -125.815,Z 145,A -96.667,B 21.9734,C -0.8443,E1 21.9769,E2 543.9968} C_DIS
LIN {X -12.9322,Y -125.4304,Z 145,A -98.625,B 21.9733,C -0.8489,E1 21.9715,E2 545.9437} C_DIS
LIN {X -16.8265,Y -124.967,Z 145,A -100.4945,B 21.9733,C -0.8456,E1 21.9663,E2 547.8237} C_DIS
LIN {X -20.1262,Y -124.479,Z 145,A -101.9562,B 21.9733,C -0.8483,E1 21.9623,E2 549.2796} C_DIS
LIN {X -24.1522,Y -123.7602,Z 145,A -103.8253,B 21.9733,C -0.8485,E1 21.9572,E2 551.1503} C_DIS
LIN {X -28.3518,Y -122.8654,Z 145,A -105.7393,B 21.9732,C -0.8511,E1 21.9519,E2 553.0603} C_DIS
LIN {X -32.3512,Y -121.8732,Z 145,A -107.5439,B 21.973,C -0.855,E1 21.9471,E2 554.8573} C_DIS
LIN {X -35.636,Y -120.9536,Z 145,A -109.1014,B 21.973,C -0.8558,E1 21.9429,E2 556.4158} C_DIS
LIN {X -39.4103,Y -119.7775,Z 145,A -111.0939,B 21.9733,C -0.849,E1 21.9375,E2 558.4306} C_DIS
LIN {X -43.538,Y -118.3411,Z 145,A -112.994,B 21.9731,C -0.8543,E1 21.9326,E2 560.3208} C_DIS
LIN {X -48.4246,Y -116.4246,Z 145,A -115.2738,B 21.9728,C -0.861,E1 21.9267,E2 562.5882} C_DIS
LIN {X -51.7167,Y -115.0002,Z 145,A -116.878,B 21.9727,C -0.8639,E1 21.9226,E2 564.1892} C_DIS
LIN {X -54.5682,Y -113.6748,Z 145,A -118.3202,B 21.9727,C -0.865,E1 21.919,E2 565.6326} C_DIS
LIN {X -57.5753,Y -112.1822,Z 145,A -119.8716,B 21.9727,C -0.8659,E1 21.9151,E2 567.1865} C_DIS
LIN {X -60.7056,Y -110.5217,Z 145,A -121.5981,B 21.9727,C -0.8632,E1 21.9108,E2 568.9258} C_DIS
LIN {X -64.362,Y -108.4328,Z 145,A -123.49,B 21.9726,C -0.8668,E1 21.9063,E2 570.8145} C_DIS
LIN {X -67.9244,Y -106.2373,Z 145,A -125.254,B 21.9723,C -0.8754,E1 21.9021,E2 572.5621} C_DIS
LIN {X -71.0209,Y -104.1934,Z 145,A -127.9314,B 21.9737,C -0.8379,E1 21.8957,E2 575.3503} C_DIS
LIN {X -76.0549,Y -100.5771,Z 145,A -129.8512,B 21.9721,C -0.879,E1 21.8916,E2 577.1678} C_DIS
LIN {X -80.1486,Y -97.3468,Z 145,A -132.1539,B 21.9719,C -0.886,E1 21.8866,E2 579.4614} C_DIS
LIN {X -82.7019,Y -95.1869,Z 145,A -133.8535,B 21.972,C -0.8817,E1 21.883,E2 581.1805} C_DIS
Enddeposition()
END
